Yaskawa INFORM job: DEMO_ROOF_UPPER_0625_3PAINT_45.JBI

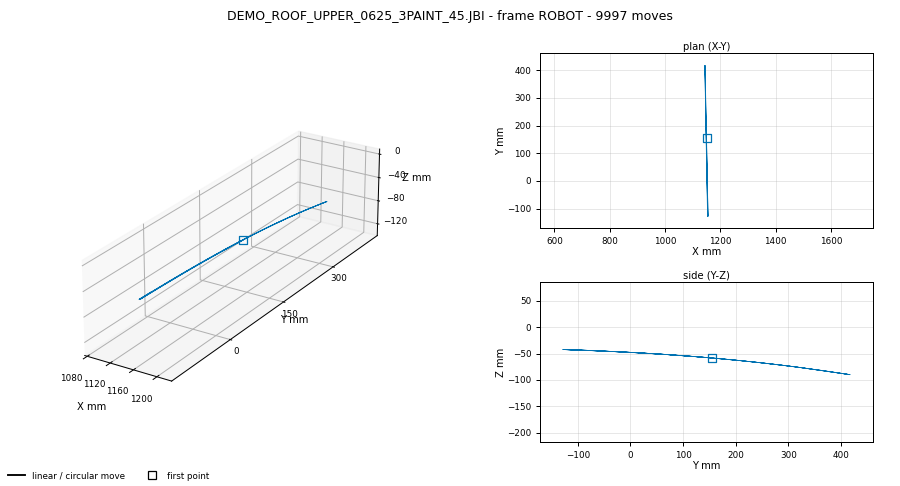
[picture p0: tool path of DEMO_ROOF_UPPER_0625_3PAINT_45.JBI in frame ROBOT, 9997 of 9997 moves have a stored position in this frame; points joined in program order, loops and branches not executed]
/JOB
//NAME DEMO_ROOF_UPPER_0625_3PAINT45
//POS
///NPOS 9997,0,0,0,0,0
///TOOL 0
///USER 0
///POSTYPE ROBOT
///RECTAN
///RCONF 1,0,0,0,0,0,0,0,0,0,0,0,0,0,0,0,0,0,0,0,0,0,0,0
C00000=1150.383,154.481,-58.197,-178.587,6.916,148.869
C00001=1150.389,154.232,-58.176,-178.590,6.914,148.870
C00002=1150.393,153.983,-58.154,-178.593,6.912,148.870
C00003=1150.398,153.733,-58.133,-178.596,6.910,148.870
C00004=1150.403,153.485,-58.111,-178.599,6.908,148.871
C00005=1150.407,153.236,-58.091,-178.601,6.907,148.871
C00006=1150.412,152.986,-58.069,-178.605,6.904,148.871
C00007=1150.417,152.737,-58.048,-178.607,6.902,148.872
C00008=1150.422,152.489,-58.026,-178.609,6.900,148.872
C00009=1150.426,152.240,-58.006,-178.612,6.899,148.872
C00010=1150.431,151.991,-57.984,-178.615,6.897,148.873
C00011=1150.436,151.741,-57.963,-178.618,6.894,148.873
C00012=1150.440,151.492,-57.941,-178.621,6.893,148.873
C00013=1150.445,151.243,-57.921,-178.624,6.891,148.874
C00014=1150.450,150.994,-57.900,-178.626,6.889,148.874
C00015=1150.455,150.745,-57.878,-178.629,6.887,148.875
C00016=1150.459,150.496,-57.857,-178.632,6.885,148.875
C00017=1150.464,150.247,-57.836,-178.635,6.883,148.875
C00018=1150.469,149.998,-57.815,-178.637,6.881,148.876
C00019=1150.473,149.749,-57.794,-178.640,6.879,148.876
C00020=1150.478,149.500,-57.773,-178.643,6.878,148.876
C00021=1150.483,149.251,-57.752,-178.645,6.876,148.877
C00022=1150.487,149.001,-57.731,-178.649,6.873,148.877
C00023=1150.492,148.752,-57.710,-178.651,6.872,148.877
C00024=1150.497,148.504,-57.688,-178.654,6.870,148.878
C00025=1150.502,148.255,-57.668,-178.657,6.868,148.878
C00026=1150.507,148.005,-57.647,-178.659,6.867,148.879
C00027=1150.511,147.756,-57.626,-178.662,6.865,148.879
C00028=1150.516,147.508,-57.605,-178.665,6.862,148.879
C00029=1150.521,147.258,-57.584,-178.668,6.860,148.879
C00030=1150.525,147.009,-57.563,-178.670,6.858,148.880
C00031=1150.530,146.760,-57.542,-178.673,6.857,148.880
C00032=1150.535,146.511,-57.522,-178.676,6.855,148.881
C00033=1150.540,146.262,-57.500,-178.679,6.853,148.881
C00034=1150.544,146.013,-57.480,-178.681,6.852,148.881
C00035=1150.549,145.764,-57.459,-178.685,6.849,148.882
C00036=1150.554,145.515,-57.438,-178.687,6.847,148.882
C00037=1150.559,145.266,-57.417,-178.690,6.846,148.883
C00038=1150.563,145.017,-57.397,-178.693,6.844,148.883
C00039=1150.568,144.767,-57.376,-178.695,6.842,148.883
C00040=1150.572,144.519,-57.355,-178.698,6.840,148.884
C00041=1150.577,144.269,-57.334,-178.701,6.839,148.884
C00042=1150.581,144.020,-57.313,-178.704,6.836,148.884
C00043=1150.587,143.771,-57.292,-178.707,6.835,148.885
C00044=1150.591,143.522,-57.272,-178.709,6.833,148.885
C00045=1150.596,143.273,-57.251,-178.712,6.831,148.885
C00046=1150.601,143.024,-57.231,-178.714,6.829,148.886
C00047=1150.606,142.774,-57.210,-178.717,6.827,148.886
C00048=1150.610,142.525,-57.189,-178.720,6.826,148.887
C00049=1150.616,142.276,-57.168,-178.723,6.823,148.887
C00050=1150.620,142.027,-57.148,-178.726,6.821,148.887
C00051=1150.624,141.778,-57.128,-178.729,6.820,148.888
C00052=1150.630,141.529,-57.107,-178.731,6.818,148.888
C00053=1150.634,141.280,-57.086,-178.734,6.816,148.889
C00054=1150.639,141.031,-57.065,-178.737,6.814,148.889
C00055=1150.644,140.782,-57.045,-178.739,6.813,148.889
C00056=1150.648,140.532,-57.025,-178.742,6.811,148.890
C00057=1150.654,140.283,-57.004,-178.745,6.809,148.890
C00058=1150.658,140.034,-56.984,-178.748,6.807,148.890
C00059=1150.662,139.785,-56.963,-178.751,6.805,148.891
C00060=1150.668,139.536,-56.943,-178.754,6.803,148.891
C00061=1150.672,139.287,-56.922,-178.756,6.802,148.892
C00062=1150.676,139.038,-56.902,-178.759,6.800,148.892
C00063=1150.682,138.789,-56.881,-178.762,6.798,148.892
C00064=1150.686,138.539,-56.861,-178.764,6.796,148.893
C00065=1150.691,138.290,-56.841,-178.767,6.795,148.893
C00066=1150.696,138.041,-56.820,-178.770,6.793,148.894
C00067=1150.700,137.792,-56.799,-178.773,6.791,148.894
C00068=1150.705,137.544,-56.779,-178.775,6.790,148.894
C00069=1150.710,137.294,-56.760,-178.779,6.787,148.895
C00070=1150.715,137.045,-56.739,-178.781,6.785,148.895
C00071=1150.720,136.796,-56.718,-178.784,6.784,148.895
C00072=1150.724,136.547,-56.698,-178.787,6.782,148.896
C00073=1150.729,136.297,-56.678,-178.789,6.780,148.896
C00074=1150.734,136.048,-56.657,-178.792,6.779,148.897
C00075=1150.739,135.799,-56.637,-178.795,6.777,148.897
C00076=1150.743,135.550,-56.617,-178.798,6.775,148.897
C00077=1150.748,135.301,-56.597,-178.800,6.773,148.898
C00078=1150.754,135.052,-56.576,-178.803,6.772,148.898
C00079=1150.758,134.803,-56.557,-178.806,6.770,148.899
C00080=1150.763,134.554,-56.536,-178.808,6.768,148.899
C00081=1150.767,134.305,-56.516,-178.811,6.767,148.899
C00082=1150.772,134.055,-56.496,-178.814,6.765,148.900
C00083=1150.776,133.806,-56.476,-178.817,6.762,148.900
C00084=1150.782,133.556,-56.456,-178.820,6.761,148.901
C00085=1150.787,133.308,-56.436,-178.823,6.759,148.901
C00086=1150.791,133.059,-56.415,-178.825,6.757,148.901
C00087=1150.796,132.810,-56.396,-178.828,6.755,148.902
C00088=1150.800,132.561,-56.375,-178.831,6.754,148.902
C00089=1150.805,132.311,-56.356,-178.833,6.752,148.903
C00090=1150.811,132.043,-56.333,-178.836,6.750,148.903
C00091=1150.815,131.774,-56.312,-178.839,6.749,148.904
C00092=1150.821,131.505,-56.291,-178.843,6.746,148.904
C00093=1150.826,131.237,-56.269,-178.845,6.745,148.904
C00094=1150.831,130.988,-56.249,-178.848,6.743,148.905
C00095=1150.836,130.739,-56.229,-178.851,6.741,148.905
C00096=1150.840,130.490,-56.209,-178.853,6.740,148.906
C00097=1150.845,130.240,-56.190,-178.856,6.738,148.906
C00098=1150.849,129.991,-56.169,-178.859,6.736,148.906
C00099=1150.856,129.742,-56.149,-178.862,6.734,148.907
C00100=1150.860,129.493,-56.129,-178.864,6.733,148.907
C00101=1150.865,129.243,-56.109,-178.867,6.731,148.907
C00102=1150.869,128.994,-56.090,-178.870,6.729,148.908
C00103=1150.874,128.746,-56.070,-178.872,6.728,148.908
C00104=1150.879,128.496,-56.050,-178.875,6.726,148.909
C00105=1150.884,128.247,-56.030,-178.878,6.724,148.909
C00106=1150.888,127.998,-56.010,-178.881,6.723,148.909
C00107=1150.894,127.749,-55.991,-178.884,6.721,148.910
C00108=1150.898,127.500,-55.970,-178.887,6.719,148.910
C00109=1150.903,127.250,-55.951,-178.889,6.718,148.911
C00110=1150.908,127.001,-55.931,-178.892,6.716,148.911
C00111=1150.912,126.752,-55.912,-178.895,6.714,148.912
C00112=1150.917,126.503,-55.892,-178.897,6.713,148.912
C00113=1150.921,126.254,-55.872,-178.900,6.711,148.912
C00114=1150.927,126.005,-55.853,-178.903,6.709,148.913
C00115=1150.931,125.756,-55.833,-178.906,6.708,148.913
C00116=1150.936,125.506,-55.813,-178.908,6.706,148.914
C00117=1150.941,125.257,-55.793,-178.911,6.704,148.914
C00118=1150.946,125.008,-55.774,-178.914,6.702,148.914
C00119=1150.951,124.758,-55.754,-178.916,6.701,148.915
C00120=1150.955,124.509,-55.734,-178.919,6.699,148.915
C00121=1150.961,124.260,-55.715,-178.922,6.698,148.916
C00122=1150.965,124.011,-55.696,-178.925,6.696,148.916
C00123=1150.969,123.762,-55.676,-178.928,6.694,148.917
C00124=1150.975,123.513,-55.657,-178.931,6.693,148.917
C00125=1150.979,123.263,-55.637,-178.933,6.691,148.917
C00126=1150.984,123.014,-55.617,-178.936,6.689,148.918
C00127=1150.989,122.765,-55.598,-178.939,6.687,148.918
C00128=1150.993,122.516,-55.578,-178.941,6.686,148.919
C00129=1150.999,122.267,-55.559,-178.944,6.684,148.919
C00130=1151.003,122.018,-55.540,-178.947,6.682,148.919
C00131=1151.008,121.768,-55.520,-178.950,6.681,148.920
C00132=1151.013,121.519,-55.501,-178.953,6.679,148.920
C00133=1151.017,121.270,-55.481,-178.955,6.678,148.921
C00134=1151.022,121.020,-55.462,-178.958,6.676,148.921
C00135=1151.027,120.771,-55.443,-178.961,6.674,148.922
C00136=1151.032,120.522,-55.423,-178.964,6.672,148.922
C00137=1151.037,120.273,-55.404,-178.966,6.671,148.923
C00138=1151.042,120.024,-55.385,-178.969,6.669,148.923
C00139=1151.047,119.775,-55.365,-178.972,6.667,148.923
C00140=1151.052,119.525,-55.346,-178.974,6.666,148.924
C00141=1151.056,119.276,-55.327,-178.977,6.664,148.924
C00142=1151.061,119.027,-55.307,-178.980,6.663,148.925
C00143=1151.066,118.778,-55.288,-178.983,6.662,148.925
C00144=1151.071,118.529,-55.268,-178.985,6.660,148.926
C00145=1151.075,118.280,-55.249,-178.988,6.658,148.926
C00146=1151.080,118.031,-55.230,-178.991,6.657,148.926
C00147=1151.085,117.781,-55.210,-178.993,6.655,148.927
C00148=1151.090,117.533,-55.192,-178.996,6.653,148.927
C00149=1151.095,117.282,-55.173,-178.999,6.651,148.928
C00150=1151.100,117.033,-55.153,-179.002,6.650,148.928
C00151=1151.104,116.784,-55.134,-179.005,6.648,148.929
C00152=1151.109,116.535,-55.115,-179.008,6.647,148.929
C00153=1151.114,116.286,-55.095,-179.010,6.645,148.929
C00154=1151.118,116.037,-55.076,-179.013,6.643,148.930
C00155=1151.124,115.787,-55.058,-179.016,6.642,148.930
C00156=1151.129,115.537,-55.038,-179.018,6.640,148.931
C00157=1151.133,115.289,-55.019,-179.021,6.639,148.931
C00158=1151.138,115.039,-55.000,-179.024,6.638,148.932
C00159=1151.143,114.791,-54.981,-179.026,6.636,148.932
C00160=1151.148,114.541,-54.962,-179.029,6.634,148.932
C00161=1151.153,114.292,-54.943,-179.032,6.633,148.933
C00162=1151.158,114.043,-54.924,-179.035,6.631,148.933
C00163=1151.162,113.794,-54.904,-179.037,6.629,148.934
C00164=1151.167,113.544,-54.886,-179.040,6.627,148.934
C00165=1151.172,113.295,-54.867,-179.043,6.626,148.935
C00166=1151.177,113.046,-54.848,-179.046,6.624,148.935
C00167=1151.182,112.796,-54.829,-179.049,6.623,148.936
C00168=1151.186,112.548,-54.810,-179.051,6.622,148.936
C00169=1151.191,112.298,-54.791,-179.054,6.620,148.936
C00170=1151.196,112.049,-54.773,-179.056,6.618,148.937
C00171=1151.201,111.800,-54.754,-179.059,6.617,148.937
C00172=1151.206,111.550,-54.734,-179.062,6.615,148.938
C00173=1151.211,111.301,-54.716,-179.065,6.614,148.938
C00174=1151.215,111.052,-54.697,-179.068,6.612,148.939
C00175=1151.221,110.802,-54.678,-179.070,6.610,148.939
C00176=1151.225,110.554,-54.660,-179.073,6.609,148.939
C00177=1151.230,110.304,-54.640,-179.075,6.608,148.940
C00178=1151.235,110.055,-54.622,-179.078,6.606,148.940
C00179=1151.240,109.806,-54.602,-179.081,6.605,148.941
C00180=1151.245,109.556,-54.584,-179.084,6.603,148.941
C00181=1151.250,109.308,-54.565,-179.087,6.601,148.942
C00182=1151.254,109.058,-54.547,-179.089,6.600,148.942
C00183=1151.260,108.809,-54.527,-179.092,6.598,148.943
C00184=1151.264,108.559,-54.509,-179.095,6.597,148.943
C00185=1151.268,108.310,-54.490,-179.097,6.596,148.944
C00186=1151.274,108.061,-54.472,-179.100,6.594,148.944
C00187=1151.278,107.812,-54.453,-179.103,6.592,148.944
C00188=1151.283,107.562,-54.435,-179.106,6.591,148.945
C00189=1151.288,107.314,-54.415,-179.108,6.589,148.945
C00190=1151.293,107.064,-54.397,-179.112,6.588,148.946
C00191=1151.298,106.814,-54.379,-179.114,6.586,148.946
C00192=1151.303,106.566,-54.360,-179.116,6.585,148.947
C00193=1151.307,106.316,-54.341,-179.119,6.583,148.947
C00194=1151.313,106.048,-54.321,-179.122,6.582,148.947
C00195=1151.318,105.780,-54.301,-179.125,6.580,148.948
C00196=1151.324,105.511,-54.281,-179.128,6.579,148.949
C00197=1151.328,105.242,-54.262,-179.132,6.576,148.949
C00198=1151.333,104.993,-54.242,-179.134,6.576,148.950
C00199=1151.338,104.744,-54.224,-179.136,6.574,148.950
C00200=1151.343,104.495,-54.206,-179.139,6.572,148.950
C00201=1151.347,104.246,-54.187,-179.142,6.571,148.951
C00202=1151.353,103.996,-54.169,-179.145,6.569,148.951
C00203=1151.358,103.747,-54.151,-179.148,6.568,148.952
C00204=1151.362,103.498,-54.132,-179.150,6.567,148.952
C00205=1151.367,103.248,-54.114,-179.153,6.565,148.953
C00206=1151.372,102.999,-54.095,-179.155,6.563,148.953
C00207=1151.377,102.750,-54.077,-179.159,6.562,148.954
C00208=1151.381,102.501,-54.058,-179.161,6.560,148.954
C00209=1151.386,102.251,-54.040,-179.164,6.559,148.955
C00210=1151.392,102.002,-54.021,-179.166,6.558,148.955
C00211=1151.397,101.753,-54.003,-179.169,6.556,148.955
C00212=1151.402,101.504,-53.986,-179.172,6.555,148.956
C00213=1151.406,101.254,-53.966,-179.175,6.553,148.956
C00214=1151.411,101.005,-53.948,-179.178,6.551,148.957
C00215=1151.416,100.756,-53.930,-179.180,6.550,148.957
C00216=1151.421,100.506,-53.912,-179.182,6.549,148.958
C00217=1151.426,100.257,-53.894,-179.186,6.547,148.958
C00218=1151.430,100.007,-53.876,-179.188,6.546,148.959
C00219=1151.435,99.758,-53.858,-179.191,6.544,148.959
C00220=1151.440,99.510,-53.839,-179.193,6.543,148.960
C00221=1151.446,99.260,-53.820,-179.196,6.541,148.960
C00222=1151.450,99.010,-53.802,-179.199,6.540,148.961
C00223=1151.455,98.761,-53.784,-179.202,6.538,148.961
C00224=1151.460,98.512,-53.766,-179.205,6.537,148.961
C00225=1151.465,98.263,-53.748,-179.207,6.536,148.962
C00226=1151.470,98.014,-53.730,-179.210,6.534,148.963
C00227=1151.474,97.764,-53.712,-179.213,6.533,148.963
C00228=1151.479,97.515,-53.694,-179.216,6.531,148.963
C00229=1151.484,97.265,-53.676,-179.218,6.529,148.964
C00230=1151.489,97.016,-53.658,-179.221,6.529,148.964
C00231=1151.494,96.767,-53.639,-179.224,6.527,148.965
C00232=1151.499,96.518,-53.621,-179.226,6.526,148.965
C00233=1151.504,96.268,-53.603,-179.229,6.524,148.966
C00234=1151.509,96.019,-53.585,-179.231,6.523,148.966
C00235=1151.513,95.769,-53.567,-179.234,6.522,148.967
C00236=1151.518,95.520,-53.549,-179.237,6.520,148.967
C00237=1151.523,95.271,-53.531,-179.240,6.518,148.968
C00238=1151.528,95.022,-53.513,-179.243,6.517,148.968
C00239=1151.533,94.773,-53.495,-179.245,6.516,148.969
C00240=1151.538,94.523,-53.477,-179.248,6.514,148.969
C00241=1151.543,94.274,-53.459,-179.251,6.513,148.969
C00242=1151.548,94.024,-53.442,-179.253,6.511,148.970
C00243=1151.553,93.775,-53.424,-179.256,6.511,148.971
C00244=1151.558,93.526,-53.406,-179.259,6.509,148.971
C00245=1151.563,93.277,-53.388,-179.261,6.507,148.971
C00246=1151.567,93.027,-53.370,-179.264,6.505,148.972
C00247=1151.572,92.778,-53.352,-179.267,6.505,148.972
C00248=1151.577,92.528,-53.334,-179.270,6.503,148.973
C00249=1151.582,92.279,-53.316,-179.272,6.502,148.973
C00250=1151.587,92.030,-53.298,-179.275,6.500,148.974
C00251=1151.591,91.781,-53.281,-179.278,6.499,148.974
C00252=1151.596,91.532,-53.263,-179.280,6.498,148.975
C00253=1151.601,91.282,-53.246,-179.283,6.496,148.975
C00254=1151.606,91.033,-53.228,-179.286,6.494,148.976
C00255=1151.611,90.784,-53.210,-179.288,6.494,148.976
C00256=1151.616,90.534,-53.192,-179.291,6.492,148.977
C00257=1151.621,90.285,-53.174,-179.294,6.490,148.977
C00258=1151.626,90.035,-53.156,-179.297,6.489,148.978
C00259=1151.631,89.786,-53.139,-179.299,6.488,148.978
C00260=1151.636,89.537,-53.122,-179.302,6.487,148.979
C00261=1151.640,89.288,-53.104,-179.305,6.485,148.979
C00262=1151.645,89.038,-53.086,-179.307,6.484,148.980
C00263=1151.650,88.789,-53.068,-179.310,6.483,148.980
C00264=1151.656,88.539,-53.051,-179.313,6.481,148.980
C00265=1151.660,88.290,-53.033,-179.316,6.479,148.981
C00266=1151.665,88.041,-53.016,-179.318,6.479,148.982
C00267=1151.670,87.792,-52.998,-179.321,6.477,148.982
C00268=1151.675,87.542,-52.980,-179.324,6.475,148.982
C00269=1151.680,87.293,-52.963,-179.327,6.474,148.983
C00270=1151.685,87.043,-52.945,-179.329,6.473,148.983
C00271=1151.689,86.794,-52.928,-179.332,6.472,148.984
C00272=1151.694,86.545,-52.910,-179.335,6.470,148.984
C00273=1151.699,86.296,-52.892,-179.337,6.469,148.985
C00274=1151.704,86.046,-52.875,-179.340,6.468,148.985
C00275=1151.709,85.797,-52.858,-179.343,6.466,148.986
C00276=1151.714,85.547,-52.840,-179.345,6.465,148.986
C00277=1151.719,85.298,-52.822,-179.348,6.464,148.987
C00278=1151.725,85.049,-52.805,-179.351,6.462,148.987
C00279=1151.729,84.800,-52.788,-179.353,6.460,148.988
C00280=1151.734,84.550,-52.771,-179.356,6.460,148.988
C00281=1151.739,84.301,-52.753,-179.359,6.458,148.989
C00282=1151.744,84.051,-52.735,-179.362,6.457,148.989
C00283=1151.748,83.802,-52.718,-179.364,6.456,148.990
C00284=1151.753,83.553,-52.701,-179.367,6.454,148.990
C00285=1151.758,83.303,-52.683,-179.370,6.453,148.991
C00286=1151.763,83.054,-52.666,-179.372,6.452,148.991
C00287=1151.768,82.804,-52.649,-179.375,6.451,148.992
C00288=1151.774,82.556,-52.631,-179.378,6.449,148.992
C00289=1151.778,82.306,-52.615,-179.380,6.448,148.993
C00290=1151.783,82.057,-52.597,-179.383,6.447,148.993
C00291=1151.788,81.807,-52.579,-179.386,6.445,148.994
C00292=1151.793,81.558,-52.563,-179.388,6.444,148.994
C00293=1151.798,81.309,-52.545,-179.391,6.443,148.995
C00294=1151.802,81.059,-52.528,-179.394,6.441,148.995
C00295=1151.808,80.810,-52.511,-179.396,6.440,148.996
C00296=1151.813,80.561,-52.493,-179.399,6.439,148.996
C00297=1151.817,80.311,-52.477,-179.402,6.437,148.997
C00298=1151.823,80.042,-52.458,-179.405,6.436,148.997
C00299=1151.829,79.774,-52.439,-179.408,6.434,148.998
C00300=1151.833,79.506,-52.421,-179.410,6.433,148.998
C00301=1151.838,79.237,-52.402,-179.413,6.432,148.999
C00302=1151.843,78.989,-52.386,-179.416,6.431,148.999
C00303=1151.849,78.739,-52.368,-179.419,6.429,149.000
C00304=1151.854,78.489,-52.351,-179.421,6.428,149.000
C00305=1151.858,78.240,-52.334,-179.424,6.427,149.001
C00306=1151.863,77.990,-52.317,-179.426,6.426,149.001
C00307=1151.868,77.742,-52.300,-179.430,6.424,149.002
C00308=1151.874,77.492,-52.283,-179.432,6.423,149.002
C00309=1151.878,77.243,-52.266,-179.434,6.422,149.003
C00310=1151.883,76.993,-52.248,-179.438,6.421,149.003
C00311=1151.887,76.744,-52.232,-179.440,6.419,149.004
C00312=1151.893,76.495,-52.215,-179.443,6.418,149.004
C00313=1151.898,76.245,-52.198,-179.446,6.417,149.005
C00314=1151.903,75.995,-52.181,-179.449,6.415,149.005
C00315=1151.907,75.746,-52.164,-179.451,6.414,149.006
C00316=1151.913,75.497,-52.147,-179.453,6.413,149.006
C00317=1151.917,75.248,-52.130,-179.456,6.412,149.007
C00318=1151.923,74.998,-52.113,-179.459,6.410,149.007
C00319=1151.927,74.749,-52.096,-179.462,6.409,149.008
C00320=1151.932,74.500,-52.080,-179.464,6.408,149.008
C00321=1151.937,74.250,-52.062,-179.467,6.407,149.009
C00322=1151.942,74.001,-52.046,-179.470,6.405,149.009
C00323=1151.948,73.751,-52.029,-179.472,6.404,149.010
C00324=1151.952,73.502,-52.012,-179.475,6.403,149.010
C00325=1151.957,73.252,-51.995,-179.477,6.402,149.011
C00326=1151.962,73.003,-51.978,-179.480,6.401,149.011
C00327=1151.967,72.754,-51.962,-179.483,6.399,149.012
C00328=1151.972,72.504,-51.945,-179.486,6.398,149.013
C00329=1151.977,72.255,-51.928,-179.489,6.397,149.013
C00330=1151.982,72.006,-51.912,-179.491,6.396,149.013
C00331=1151.987,71.756,-51.894,-179.494,6.395,149.014
C00332=1151.991,71.507,-51.878,-179.497,6.393,149.014
C00333=1151.997,71.258,-51.861,-179.499,6.392,149.015
C00334=1152.002,71.008,-51.844,-179.502,6.391,149.016
C00335=1152.006,70.759,-51.827,-179.504,6.390,149.016
C00336=1152.011,70.510,-51.811,-179.507,6.388,149.016
C00337=1152.017,70.260,-51.794,-179.510,6.387,149.017
C00338=1152.021,70.010,-51.777,-179.512,6.386,149.017
C00339=1152.026,69.762,-51.761,-179.515,6.384,149.018
C00340=1152.031,69.512,-51.744,-179.518,6.384,149.019
C00341=1152.036,69.262,-51.728,-179.520,6.382,149.019
C00342=1152.041,69.013,-51.711,-179.523,6.381,149.019
C00343=1152.046,68.763,-51.694,-179.526,6.380,149.020
C00344=1152.051,68.514,-51.678,-179.529,6.378,149.021
C00345=1152.056,68.265,-51.661,-179.531,6.378,149.021
C00346=1152.060,68.015,-51.644,-179.534,6.376,149.022
C00347=1152.067,67.766,-51.628,-179.536,6.375,149.022
C00348=1152.071,67.516,-51.612,-179.539,6.374,149.023
C00349=1152.076,67.267,-51.595,-179.542,6.372,149.023
C00350=1152.081,67.018,-51.579,-179.544,6.372,149.024
C00351=1152.086,66.768,-51.561,-179.547,6.370,149.024
C00352=1152.091,66.519,-51.546,-179.550,6.369,149.025
C00353=1152.096,66.269,-51.529,-179.552,6.368,149.025
C00354=1152.100,66.020,-51.512,-179.555,6.367,149.026
C00355=1152.105,65.771,-51.496,-179.558,6.366,149.026
C00356=1152.111,65.521,-51.480,-179.560,6.364,149.027
C00357=1152.116,65.272,-51.463,-179.563,6.363,149.027
C00358=1152.120,65.022,-51.447,-179.566,6.362,149.028
C00359=1152.125,64.774,-51.430,-179.568,6.361,149.028
C00360=1152.130,64.523,-51.414,-179.571,6.360,149.029
C00361=1152.135,64.275,-51.398,-179.573,6.359,149.029
C00362=1152.140,64.025,-51.381,-179.577,6.357,149.030
C00363=1152.145,63.775,-51.365,-179.579,6.357,149.030
C00364=1152.150,63.526,-51.349,-179.581,6.355,149.031
C00365=1152.155,63.276,-51.333,-179.585,6.354,149.031
C00366=1152.160,63.027,-51.316,-179.587,6.353,149.032
C00367=1152.165,62.778,-51.300,-179.590,6.351,149.032
C00368=1152.170,62.528,-51.284,-179.592,6.351,149.033
C00369=1152.175,62.279,-51.267,-179.595,6.349,149.033
C00370=1152.180,62.030,-51.251,-179.598,6.348,149.034
C00371=1152.185,61.780,-51.235,-179.600,6.347,149.035
C00372=1152.190,61.531,-51.218,-179.602,6.346,149.035
C00373=1152.195,61.281,-51.202,-179.606,6.345,149.036
C00374=1152.200,61.032,-51.186,-179.608,6.344,149.036
C00375=1152.205,60.782,-51.170,-179.611,6.342,149.037
C00376=1152.210,60.533,-51.154,-179.613,6.342,149.037
C00377=1152.215,60.283,-51.138,-179.616,6.340,149.038
C00378=1152.220,60.034,-51.121,-179.619,6.339,149.038
C00379=1152.225,59.784,-51.105,-179.621,6.338,149.039
C00380=1152.230,59.535,-51.089,-179.624,6.336,149.039
C00381=1152.235,59.286,-51.074,-179.627,6.336,149.040
C00382=1152.240,59.036,-51.057,-179.629,6.334,149.040
C00383=1152.245,58.787,-51.041,-179.632,6.334,149.041
C00384=1152.249,58.537,-51.025,-179.635,6.332,149.041
C00385=1152.255,58.288,-51.009,-179.637,6.331,149.042
C00386=1152.259,58.039,-50.992,-179.640,6.330,149.042
C00387=1152.265,57.789,-50.977,-179.642,6.329,149.043
C00388=1152.270,57.539,-50.961,-179.646,6.328,149.044
C00389=1152.275,57.290,-50.945,-179.648,6.327,149.044
C00390=1152.280,57.041,-50.929,-179.651,6.325,149.044
C00391=1152.284,56.791,-50.912,-179.653,6.325,149.045
C00392=1152.290,56.542,-50.897,-179.656,6.323,149.046
C00393=1152.295,56.292,-50.881,-179.658,6.322,149.046
C00394=1152.300,56.043,-50.864,-179.661,6.321,149.047
C00395=1152.305,55.794,-50.849,-179.663,6.320,149.047
C00396=1152.310,55.544,-50.833,-179.667,6.319,149.048
C00397=1152.315,55.295,-50.817,-179.669,6.318,149.048
C00398=1152.319,55.045,-50.801,-179.672,6.316,149.049
C00399=1152.324,54.796,-50.786,-179.674,6.316,149.049
C00400=1152.329,54.547,-50.769,-179.677,6.314,149.050
C00401=1152.334,54.297,-50.753,-179.680,6.313,149.050
C00402=1152.340,54.028,-50.736,-179.682,6.312,149.051
C00403=1152.345,53.760,-50.719,-179.685,6.311,149.052
C00404=1152.351,53.491,-50.702,-179.688,6.310,149.052
C00405=1152.356,53.223,-50.685,-179.691,6.308,149.053
C00406=1152.361,52.973,-50.669,-179.693,6.308,149.053
C00407=1152.367,52.723,-50.654,-179.696,6.306,149.054
C00408=1152.371,52.475,-50.638,-179.699,6.305,149.054
C00409=1152.376,52.225,-50.622,-179.702,6.304,149.055
C00410=1152.381,51.975,-50.607,-179.704,6.303,149.055
C00411=1152.387,51.726,-50.591,-179.706,6.302,149.056
C00412=1152.391,51.476,-50.575,-179.709,6.301,149.056
C00413=1152.396,51.227,-50.559,-179.711,6.300,149.057
C00414=1152.401,50.978,-50.544,-179.715,6.299,149.058
C00415=1152.406,50.728,-50.528,-179.717,6.298,149.058
C00416=1152.411,50.478,-50.512,-179.720,6.297,149.058
C00417=1152.417,50.229,-50.497,-179.722,6.296,149.059
C00418=1152.421,49.979,-50.481,-179.725,6.294,149.060
C00419=1152.426,49.730,-50.466,-179.728,6.294,149.060
C00420=1152.431,49.481,-50.449,-179.730,6.292,149.061
C00421=1152.437,49.232,-50.434,-179.733,6.292,149.061
C00422=1152.441,48.982,-50.418,-179.735,6.291,149.062
C00423=1152.446,48.732,-50.403,-179.738,6.289,149.062
C00424=1152.451,48.483,-50.387,-179.741,6.289,149.063
C00425=1152.456,48.233,-50.371,-179.743,6.287,149.063
C00426=1152.461,47.984,-50.356,-179.746,6.287,149.064
C00427=1152.466,47.734,-50.341,-179.749,6.285,149.064
C00428=1152.472,47.485,-50.325,-179.751,6.284,149.065
C00429=1152.476,47.235,-50.310,-179.754,6.283,149.066
C00430=1152.481,46.986,-50.294,-179.756,6.282,149.066
C00431=1152.486,46.736,-50.279,-179.759,6.282,149.067
C00432=1152.491,46.487,-50.264,-179.762,6.280,149.067
C00433=1152.496,46.238,-50.248,-179.764,6.279,149.068
C00434=1152.501,45.988,-50.232,-179.767,6.278,149.068
C00435=1152.506,45.739,-50.217,-179.769,6.277,149.069
C00436=1152.511,45.489,-50.201,-179.772,6.276,149.069
C00437=1152.517,45.240,-50.186,-179.775,6.275,149.070
C00438=1152.521,44.990,-50.171,-179.777,6.274,149.070
C00439=1152.526,44.741,-50.155,-179.780,6.273,149.071
C00440=1152.531,44.491,-50.139,-179.783,6.272,149.072
C00441=1152.536,44.242,-50.124,-179.785,6.271,149.072
C00442=1152.541,43.993,-50.109,-179.788,6.270,149.072
C00443=1152.546,43.742,-50.094,-179.790,6.269,149.073
C00444=1152.551,43.493,-50.079,-179.793,6.268,149.074
C00445=1152.557,43.244,-50.063,-179.796,6.267,149.074
C00446=1152.561,42.995,-50.048,-179.798,6.265,149.075
C00447=1152.567,42.745,-50.032,-179.801,6.265,149.075
C00448=1152.571,42.496,-50.017,-179.803,6.264,149.076
C00449=1152.576,42.246,-50.001,-179.806,6.262,149.076
C00450=1152.582,41.996,-49.987,-179.809,6.262,149.077
C00451=1152.586,41.747,-49.972,-179.811,6.260,149.077
C00452=1152.592,41.497,-49.956,-179.814,6.260,149.078
C00453=1152.596,41.248,-49.941,-179.816,6.259,149.078
C00454=1152.602,40.999,-49.925,-179.819,6.258,149.079
C00455=1152.607,40.749,-49.911,-179.821,6.257,149.080
C00456=1152.612,40.499,-49.895,-179.825,6.256,149.080
C00457=1152.616,40.250,-49.880,-179.827,6.255,149.081
C00458=1152.622,40.001,-49.865,-179.829,6.254,149.081
C00459=1152.627,39.751,-49.850,-179.832,6.253,149.082
C00460=1152.632,39.502,-49.835,-179.834,6.252,149.082
C00461=1152.637,39.252,-49.820,-179.838,6.251,149.083
C00462=1152.642,39.003,-49.804,-179.840,6.250,149.083
C00463=1152.647,38.753,-49.790,-179.842,6.249,149.084
C00464=1152.652,38.504,-49.774,-179.845,6.248,149.085
C00465=1152.657,38.255,-49.759,-179.847,6.247,149.085
C00466=1152.662,38.004,-49.744,-179.850,6.246,149.086
C00467=1152.667,37.755,-49.729,-179.853,6.245,149.086
C00468=1152.672,37.506,-49.713,-179.855,6.244,149.087
C00469=1152.677,37.256,-49.699,-179.858,6.243,149.087
C00470=1152.682,37.006,-49.684,-179.861,6.242,149.088
C00471=1152.687,36.757,-49.669,-179.863,6.241,149.088
C00472=1152.692,36.508,-49.654,-179.866,6.240,149.089
C00473=1152.697,36.258,-49.639,-179.868,6.239,149.089
C00474=1152.702,36.009,-49.624,-179.871,6.238,149.090
C00475=1152.708,35.759,-49.609,-179.874,6.237,149.091
C00476=1152.713,35.509,-49.595,-179.876,6.236,149.091
C00477=1152.717,35.260,-49.580,-179.879,6.236,149.092
C00478=1152.723,35.011,-49.564,-179.881,6.234,149.092
C00479=1152.728,34.761,-49.550,-179.884,6.234,149.093
C00480=1152.733,34.512,-49.534,-179.886,6.233,149.093
C00481=1152.738,34.262,-49.520,-179.889,6.231,149.094
C00482=1152.743,34.013,-49.505,-179.892,6.231,149.094
C00483=1152.748,33.763,-49.490,-179.895,6.229,149.095
C00484=1152.753,33.514,-49.475,-179.897,6.229,149.096
C00485=1152.758,33.264,-49.461,-179.899,6.228,149.096
C00486=1152.763,33.015,-49.445,-179.902,6.226,149.097
C00487=1152.768,32.765,-49.431,-179.905,6.226,149.097
C00488=1152.773,32.516,-49.416,-179.907,6.225,149.098
C00489=1152.779,32.266,-49.401,-179.910,6.223,149.098
C00490=1152.783,32.017,-49.386,-179.913,6.223,149.099
C00491=1152.788,31.767,-49.372,-179.915,6.222,149.099
C00492=1152.793,31.518,-49.357,-179.918,6.221,149.100
C00493=1152.799,31.268,-49.342,-179.920,6.220,149.100
C00494=1152.804,31.018,-49.328,-179.923,6.220,149.101
C00495=1152.808,30.769,-49.313,-179.926,6.218,149.102
C00496=1152.814,30.519,-49.298,-179.928,6.217,149.102
C00497=1152.819,30.270,-49.283,-179.930,6.217,149.103
C00498=1152.824,30.020,-49.268,-179.933,6.216,149.103
C00499=1152.829,29.771,-49.254,-179.936,6.215,149.104
C00500=1152.834,29.521,-49.239,-179.938,6.214,149.104
C00501=1152.839,29.272,-49.224,-179.941,6.213,149.105
C00502=1152.844,29.022,-49.210,-179.943,6.212,149.105
C00503=1152.848,28.773,-49.195,-179.946,6.211,149.106
C00504=1152.854,28.524,-49.181,-179.948,6.210,149.107
C00505=1152.860,28.274,-49.166,-179.951,6.209,149.107
C00506=1152.865,28.005,-49.151,-179.954,6.208,149.108
C00507=1152.870,27.736,-49.135,-179.957,6.207,149.108
C00508=1152.876,27.467,-49.119,-179.959,6.207,149.109
C00509=1152.881,27.198,-49.103,-179.962,6.205,149.110
C00510=1152.886,26.949,-49.089,-179.965,6.204,149.110
C00511=1152.891,26.699,-49.074,-179.967,6.204,149.111
C00512=1152.896,26.449,-49.060,-179.970,6.202,149.111
C00513=1152.901,26.200,-49.044,-179.972,6.201,149.112
C00514=1152.907,25.951,-49.030,-179.975,6.201,149.112
C00515=1152.912,25.701,-49.016,-179.977,6.200,149.113
C00516=1152.917,25.451,-49.002,-179.980,6.199,149.113
C00517=1152.922,25.202,-48.988,-179.983,6.198,149.114
C00518=1152.926,24.953,-48.973,-179.985,6.197,149.115
C00519=1152.931,24.703,-48.958,-179.988,6.196,149.115
C00520=1152.936,24.453,-48.944,-179.990,6.195,149.116
C00521=1152.942,24.204,-48.930,-179.993,6.195,149.116
C00522=1152.947,23.954,-48.915,-179.995,6.194,149.117
C00523=1152.952,23.705,-48.900,-179.998,6.193,149.117
C00524=1152.957,23.455,-48.886,180.000,6.192,149.118
C00525=1152.962,23.206,-48.872,179.997,6.191,149.119
C00526=1152.967,22.956,-48.858,179.994,6.190,149.119
C00527=1152.972,22.706,-48.843,179.991,6.189,149.120
C00528=1152.977,22.457,-48.829,179.989,6.188,149.120
C00529=1152.982,22.207,-48.815,179.987,6.188,149.121
C00530=1152.987,21.958,-48.801,179.984,6.186,149.121
C00531=1152.992,21.708,-48.786,179.982,6.185,149.122
C00532=1152.997,21.458,-48.772,179.979,6.185,149.122
C00533=1153.003,21.210,-48.758,179.977,6.184,149.123
C00534=1153.007,20.960,-48.743,179.974,6.183,149.124
C00535=1153.012,20.711,-48.729,179.972,6.182,149.124
C00536=1153.017,20.461,-48.715,179.969,6.182,149.125
C00537=1153.022,20.211,-48.700,179.967,6.181,149.125
C00538=1153.028,19.962,-48.687,179.963,6.180,149.126
C00539=1153.033,19.712,-48.672,179.961,6.179,149.126
C00540=1153.038,19.463,-48.658,179.959,6.178,149.127
C00541=1153.043,19.213,-48.644,179.956,6.177,149.127
C00542=1153.048,18.964,-48.630,179.953,6.176,149.128
C00543=1153.053,18.714,-48.616,179.951,6.175,149.129
C00544=1153.058,18.465,-48.601,179.948,6.175,149.129
C00545=1153.063,18.215,-48.587,179.946,6.174,149.130
C00546=1153.069,17.966,-48.573,179.943,6.173,149.130
C00547=1153.074,17.715,-48.560,179.941,6.172,149.131
C00548=1153.079,17.466,-48.545,179.938,6.172,149.132
C00549=1153.084,17.216,-48.531,179.936,6.171,149.132
C00550=1153.089,16.967,-48.517,179.933,6.169,149.133
C00551=1153.094,16.717,-48.503,179.931,6.169,149.133
C00552=1153.099,16.468,-48.488,179.928,6.168,149.134
C00553=1153.104,16.218,-48.474,179.926,6.167,149.134
C00554=1153.110,15.969,-48.460,179.923,6.166,149.135
C00555=1153.114,15.720,-48.447,179.920,6.165,149.135
C00556=1153.119,15.470,-48.432,179.918,6.164,149.136
C00557=1153.125,15.220,-48.419,179.916,6.164,149.137
C00558=1153.130,14.970,-48.405,179.913,6.163,149.137
C00559=1153.135,14.721,-48.391,179.910,6.162,149.138
C00560=1153.140,14.472,-48.377,179.908,6.161,149.138
C00561=1153.145,14.222,-48.362,179.905,6.161,149.139
C00562=1153.150,13.973,-48.349,179.903,6.160,149.139
C00563=1153.155,13.723,-48.336,179.900,6.159,149.140
C00564=1153.160,13.473,-48.321,179.898,6.158,149.140
C00565=1153.165,13.224,-48.307,179.895,6.157,149.141
C00566=1153.171,12.975,-48.293,179.893,6.156,149.142
C00567=1153.176,12.724,-48.280,179.890,6.156,149.142
C00568=1153.180,12.475,-48.266,179.887,6.154,149.143
C00569=1153.186,12.226,-48.252,179.885,6.154,149.143
C00570=1153.191,11.976,-48.238,179.883,6.153,149.144
C00571=1153.196,11.726,-48.224,179.880,6.153,149.145
C00572=1153.202,11.477,-48.210,179.878,6.152,149.145
C00573=1153.206,11.227,-48.196,179.875,6.151,149.146
C00574=1153.211,10.977,-48.183,179.872,6.150,149.146
C00575=1153.217,10.728,-48.169,179.870,6.149,149.147
C00576=1153.222,10.478,-48.155,179.868,6.148,149.147
C00577=1153.227,10.229,-48.141,179.865,6.148,149.148
C00578=1153.232,9.979,-48.128,179.862,6.146,149.148
C00579=1153.237,9.730,-48.114,179.860,6.146,149.149
C00580=1153.242,9.481,-48.100,179.857,6.145,149.150
C00581=1153.247,9.231,-48.087,179.855,6.144,149.150
C00582=1153.252,8.982,-48.073,179.853,6.144,149.151
C00583=1153.258,8.731,-48.059,179.850,6.142,149.151
C00584=1153.263,8.482,-48.045,179.847,6.142,149.152
C00585=1153.267,8.233,-48.032,179.845,6.141,149.152
C00586=1153.273,7.982,-48.018,179.842,6.140,149.153
C00587=1153.278,7.733,-48.004,179.840,6.140,149.154
C00588=1153.283,7.483,-47.991,179.837,6.139,149.154
C00589=1153.288,7.234,-47.977,179.835,6.138,149.155
C00590=1153.293,6.985,-47.963,179.832,6.137,149.155
C00591=1153.298,6.735,-47.950,179.830,6.136,149.156
C00592=1153.303,6.486,-47.936,179.827,6.136,149.157
C00593=1153.309,6.235,-47.923,179.825,6.135,149.157
C00594=1153.313,5.987,-47.909,179.822,6.135,149.158
C00595=1153.319,5.736,-47.896,179.820,6.133,149.158
C00596=1153.324,5.487,-47.882,179.817,6.133,149.159
C00597=1153.329,5.237,-47.869,179.815,6.132,149.159
C00598=1153.334,4.988,-47.855,179.812,6.131,149.160
C00599=1153.340,4.738,-47.841,179.810,6.130,149.160
C00600=1153.344,4.489,-47.828,179.807,6.130,149.161
C00601=1153.350,4.239,-47.814,179.805,6.128,149.162
C00602=1153.354,3.990,-47.801,179.802,6.128,149.162
C00603=1153.360,3.740,-47.788,179.800,6.127,149.163
C00604=1153.365,3.490,-47.773,179.797,6.127,149.163
C00605=1153.370,3.241,-47.761,179.795,6.126,149.164
C00606=1153.375,2.991,-47.747,179.792,6.125,149.165
C00607=1153.380,2.742,-47.734,179.790,6.125,149.165
C00608=1153.385,2.492,-47.720,179.787,6.123,149.166
C00609=1153.391,2.243,-47.706,179.785,6.123,149.166
C00610=1153.396,1.973,-47.693,179.782,6.122,149.167
C00611=1153.401,1.703,-47.678,179.779,6.122,149.168
C00612=1153.407,1.434,-47.664,179.777,6.120,149.168
C00613=1153.412,1.165,-47.649,179.774,6.120,149.169
C00614=1153.418,0.915,-47.636,179.772,6.119,149.169
C00615=1153.422,0.666,-47.622,179.769,6.118,149.170
C00616=1153.428,0.416,-47.609,179.767,6.118,149.170
C00617=1153.433,0.166,-47.596,179.764,6.116,149.171
C00618=1153.438,-0.083,-47.582,179.761,6.115,149.171
C00619=1153.443,-0.333,-47.569,179.759,6.115,149.172
C00620=1153.449,-0.582,-47.556,179.757,6.114,149.173
C00621=1153.454,-0.832,-47.542,179.754,6.114,149.173
C00622=1153.459,-1.081,-47.529,179.752,6.113,149.174
C00623=1153.464,-1.331,-47.516,179.749,6.113,149.174
C00624=1153.469,-1.581,-47.503,179.747,6.112,149.175
C00625=1153.474,-1.830,-47.490,179.744,6.110,149.176
C00626=1153.479,-2.080,-47.476,179.742,6.110,149.176
C00627=1153.484,-2.329,-47.464,179.739,6.109,149.177
C00628=1153.489,-2.580,-47.450,179.737,6.108,149.177
C00629=1153.494,-2.828,-47.437,179.734,6.108,149.178
C00630=1153.500,-3.078,-47.424,179.732,6.107,149.178
C00631=1153.505,-3.328,-47.411,179.729,6.107,149.179
C00632=1153.511,-3.578,-47.397,179.727,6.106,149.180
C00633=1153.515,-3.828,-47.385,179.724,6.105,149.180
C00634=1153.520,-4.076,-47.371,179.722,6.104,149.181
C00635=1153.526,-4.326,-47.358,179.719,6.103,149.181
C00636=1153.530,-4.576,-47.345,179.717,6.103,149.182
C00637=1153.536,-4.826,-47.332,179.714,6.102,149.183
C00638=1153.541,-5.075,-47.319,179.712,6.101,149.183
C00639=1153.546,-5.325,-47.306,179.709,6.101,149.184
C00640=1153.552,-5.575,-47.293,179.707,6.100,149.184
C00641=1153.556,-5.824,-47.279,179.704,6.100,149.185
C00642=1153.561,-6.073,-47.267,179.702,6.099,149.185
C00643=1153.567,-6.323,-47.254,179.700,6.098,149.186
C00644=1153.571,-6.573,-47.241,179.697,6.097,149.186
C00645=1153.577,-6.823,-47.227,179.694,6.096,149.187
C00646=1153.582,-7.072,-47.215,179.692,6.096,149.188
C00647=1153.587,-7.322,-47.202,179.689,6.095,149.188
C00648=1153.593,-7.572,-47.189,179.687,6.094,149.189
C00649=1153.598,-7.821,-47.176,179.685,6.094,149.189
C00650=1153.602,-8.071,-47.163,179.682,6.093,149.190
C00651=1153.608,-8.320,-47.151,179.680,6.093,149.191
C00652=1153.613,-8.570,-47.137,179.678,6.092,149.191
C00653=1153.618,-8.820,-47.124,179.675,6.091,149.192
C00654=1153.623,-9.069,-47.111,179.673,6.091,149.192
C00655=1153.629,-9.318,-47.098,179.670,6.090,149.193
C00656=1153.634,-9.568,-47.085,179.667,6.089,149.193
C00657=1153.638,-9.818,-47.072,179.665,6.088,149.194
C00658=1153.643,-10.067,-47.060,179.662,6.087,149.195
C00659=1153.650,-10.317,-47.047,179.660,6.087,149.195
C00660=1153.654,-10.567,-47.034,179.658,6.086,149.196
C00661=1153.659,-10.816,-47.022,179.655,6.086,149.196
C00662=1153.664,-11.066,-47.009,179.653,6.085,149.197
C00663=1153.670,-11.315,-46.996,179.650,6.084,149.198
C00664=1153.675,-11.565,-46.983,179.648,6.084,149.198
C00665=1153.680,-11.815,-46.970,179.645,6.083,149.199
C00666=1153.685,-12.064,-46.958,179.643,6.082,149.199
C00667=1153.690,-12.314,-46.944,179.641,6.081,149.200
C00668=1153.695,-12.564,-46.932,179.638,6.081,149.200
C00669=1153.700,-12.813,-46.919,179.636,6.080,149.201
C00670=1153.706,-13.062,-46.906,179.633,6.080,149.202
C00671=1153.710,-13.312,-46.893,179.631,6.079,149.202
C00672=1153.716,-13.563,-46.881,179.629,6.079,149.203
C00673=1153.721,-13.812,-46.868,179.626,6.077,149.203
C00674=1153.726,-14.061,-46.856,179.623,6.077,149.204
C00675=1153.732,-14.311,-46.843,179.621,6.076,149.204
C00676=1153.736,-14.561,-46.830,179.618,6.075,149.205
C00677=1153.741,-14.810,-46.817,179.616,6.074,149.205
C00678=1153.747,-15.060,-46.805,179.613,6.074,149.206
C00679=1153.753,-15.309,-46.792,179.611,6.073,149.207
C00680=1153.757,-15.560,-46.779,179.609,6.073,149.207
C00681=1153.762,-15.809,-46.767,179.606,6.072,149.208
C00682=1153.767,-16.058,-46.754,179.604,6.072,149.209
C00683=1153.773,-16.308,-46.742,179.602,6.071,149.209
C00684=1153.778,-16.557,-46.730,179.599,6.070,149.210
C00685=1153.782,-16.807,-46.717,179.597,6.070,149.210
C00686=1153.788,-17.057,-46.704,179.594,6.069,149.211
C00687=1153.794,-17.307,-46.692,179.592,6.068,149.211
C00688=1153.799,-17.556,-46.679,179.589,6.068,149.212
C00689=1153.804,-17.806,-46.667,179.587,6.067,149.212
C00690=1153.809,-18.055,-46.654,179.584,6.067,149.213
C00691=1153.814,-18.306,-46.642,179.582,6.066,149.214
C00692=1153.819,-18.555,-46.629,179.580,6.065,149.214
C00693=1153.824,-18.804,-46.616,179.577,6.065,149.215
C00694=1153.830,-19.054,-46.605,179.575,6.064,149.215
C00695=1153.835,-19.303,-46.592,179.573,6.063,149.216
C00696=1153.840,-19.553,-46.579,179.570,6.063,149.217
C00697=1153.845,-19.803,-46.567,179.568,6.062,149.217
C00698=1153.850,-20.053,-46.555,179.565,6.062,149.218
C00699=1153.855,-20.302,-46.542,179.563,6.061,149.218
C00700=1153.860,-20.552,-46.530,179.560,6.060,149.219
C00701=1153.866,-20.802,-46.517,179.558,6.060,149.219
C00702=1153.871,-21.051,-46.504,179.555,6.059,149.220
C00703=1153.877,-21.301,-46.492,179.553,6.058,149.221
C00704=1153.882,-21.550,-46.480,179.551,6.058,149.221
C00705=1153.887,-21.800,-46.468,179.548,6.057,149.222
C00706=1153.892,-22.049,-46.455,179.546,6.057,149.222
C00707=1153.897,-22.299,-46.442,179.544,6.056,149.223
C00708=1153.902,-22.549,-46.430,179.541,6.056,149.224
C00709=1153.907,-22.799,-46.418,179.539,6.055,149.224
C00710=1153.912,-23.048,-46.407,179.536,6.054,149.225
C00711=1153.917,-23.298,-46.394,179.534,6.054,149.225
C00712=1153.923,-23.548,-46.382,179.531,6.053,149.226
C00713=1153.928,-23.797,-46.369,179.529,6.052,149.226
C00714=1153.934,-24.068,-46.356,179.526,6.052,149.227
C00715=1153.939,-24.337,-46.343,179.524,6.050,149.228
C00716=1153.945,-24.607,-46.330,179.521,6.050,149.228
C00717=1153.950,-24.877,-46.317,179.518,6.049,149.229
C00718=1153.955,-25.127,-46.304,179.516,6.049,149.229
C00719=1153.961,-25.377,-46.292,179.513,6.048,149.230
C00720=1153.966,-25.626,-46.280,179.511,6.047,149.231
C00721=1153.971,-25.876,-46.268,179.509,6.047,149.231
C00722=1153.976,-26.125,-46.255,179.506,6.046,149.232
C00723=1153.982,-26.375,-46.243,179.504,6.046,149.233
C00724=1153.987,-26.624,-46.231,179.502,6.045,149.233
C00725=1153.992,-26.874,-46.219,179.499,6.045,149.234
C00726=1153.997,-27.123,-46.207,179.497,6.044,149.234
C00727=1154.002,-27.373,-46.195,179.494,6.043,149.235
C00728=1154.008,-27.623,-46.183,179.492,6.043,149.235
C00729=1154.013,-27.873,-46.170,179.489,6.042,149.236
C00730=1154.018,-28.122,-46.158,179.487,6.041,149.237
C00731=1154.023,-28.372,-46.146,179.485,6.042,149.237
C00732=1154.029,-28.622,-46.134,179.483,6.041,149.238
C00733=1154.033,-28.871,-46.123,179.480,6.040,149.238
C00734=1154.038,-29.121,-46.110,179.478,6.040,149.239
C00735=1154.044,-29.371,-46.098,179.476,6.039,149.239
C00736=1154.049,-29.621,-46.086,179.473,6.038,149.240
C00737=1154.054,-29.870,-46.074,179.471,6.038,149.240
C00738=1154.059,-30.119,-46.062,179.468,6.037,149.241
C00739=1154.065,-30.369,-46.050,179.466,6.036,149.242
C00740=1154.070,-30.619,-46.038,179.463,6.036,149.242
C00741=1154.075,-30.869,-46.026,179.461,6.035,149.243
C00742=1154.081,-31.119,-46.014,179.459,6.035,149.244
C00743=1154.085,-31.368,-46.002,179.456,6.034,149.244
C00744=1154.090,-31.618,-45.990,179.454,6.034,149.245
C00745=1154.096,-31.867,-45.978,179.451,6.033,149.245
C00746=1154.101,-32.117,-45.966,179.449,6.032,149.246
C00747=1154.106,-32.366,-45.954,179.447,6.032,149.246
C00748=1154.111,-32.616,-45.943,179.444,6.031,149.247
C00749=1154.116,-32.866,-45.931,179.442,6.030,149.248
C00750=1154.122,-33.116,-45.918,179.439,6.030,149.248
C00751=1154.127,-33.365,-45.907,179.438,6.030,149.249
C00752=1154.132,-33.614,-45.895,179.435,6.030,149.249
C00753=1154.138,-33.864,-45.883,179.433,6.029,149.250
C00754=1154.143,-34.114,-45.872,179.430,6.028,149.251
C00755=1154.148,-34.363,-45.860,179.428,6.027,149.251
C00756=1154.153,-34.613,-45.848,179.425,6.027,149.252
C00757=1154.158,-34.863,-45.836,179.423,6.026,149.252
C00758=1154.163,-35.113,-45.824,179.421,6.025,149.253
C00759=1154.169,-35.363,-45.813,179.418,6.025,149.253
C00760=1154.174,-35.613,-45.801,179.416,6.024,149.254
C00761=1154.178,-35.862,-45.789,179.413,6.024,149.255
C00762=1154.184,-36.111,-45.777,179.411,6.023,149.255
C00763=1154.190,-36.361,-45.765,179.408,6.023,149.256
C00764=1154.195,-36.611,-45.753,179.406,6.022,149.256
C00765=1154.200,-36.860,-45.742,179.404,6.022,149.257
C00766=1154.205,-37.110,-45.730,179.402,6.021,149.257
C00767=1154.210,-37.360,-45.719,179.399,6.021,149.258
C00768=1154.216,-37.610,-45.707,179.397,6.020,149.259
C00769=1154.221,-37.859,-45.694,179.395,6.020,149.259
C00770=1154.226,-38.108,-45.684,179.392,6.019,149.260
C00771=1154.231,-38.358,-45.672,179.390,6.019,149.260
C00772=1154.237,-38.608,-45.660,179.387,6.018,149.261
C00773=1154.241,-38.858,-45.648,179.385,6.017,149.262
C00774=1154.247,-39.108,-45.637,179.383,6.017,149.262
C00775=1154.252,-39.358,-45.625,179.380,6.016,149.263
C00776=1154.258,-39.606,-45.614,179.378,6.016,149.263
C00777=1154.263,-39.856,-45.602,179.376,6.015,149.264
C00778=1154.268,-40.106,-45.591,179.374,6.015,149.264
C00779=1154.273,-40.356,-45.579,179.371,6.014,149.265
C00780=1154.278,-40.606,-45.567,179.369,6.014,149.266
C00781=1154.283,-40.856,-45.556,179.366,6.013,149.266
C00782=1154.289,-41.105,-45.544,179.364,6.013,149.267
C00783=1154.294,-41.354,-45.533,179.362,6.012,149.267
C00784=1154.299,-41.604,-45.521,179.359,6.011,149.268
C00785=1154.304,-41.854,-45.510,179.357,6.011,149.268
C00786=1154.310,-42.104,-45.498,179.355,6.011,149.269
C00787=1154.315,-42.353,-45.487,179.353,6.010,149.270
C00788=1154.320,-42.603,-45.475,179.350,6.010,149.270
C00789=1154.325,-42.852,-45.464,179.348,6.009,149.271
C00790=1154.330,-43.102,-45.452,179.346,6.008,149.271
C00791=1154.335,-43.352,-45.440,179.343,6.008,149.272
C00792=1154.341,-43.602,-45.430,179.341,6.007,149.272
C00793=1154.346,-43.851,-45.418,179.338,6.007,149.273
C00794=1154.352,-44.101,-45.406,179.336,6.007,149.274
C00795=1154.356,-44.351,-45.395,179.334,6.006,149.274
C00796=1154.362,-44.600,-45.384,179.332,6.005,149.275
C00797=1154.367,-44.850,-45.372,179.329,6.005,149.275
C00798=1154.372,-45.100,-45.360,179.327,6.004,149.276
C00799=1154.377,-45.349,-45.349,179.324,6.004,149.277
C00800=1154.383,-45.599,-45.337,179.322,6.003,149.277
C00801=1154.388,-45.849,-45.327,179.320,6.002,149.278
C00802=1154.394,-46.099,-45.315,179.318,6.003,149.278
C00803=1154.398,-46.348,-45.304,179.315,6.002,149.279
C00804=1154.404,-46.598,-45.292,179.313,6.001,149.280
C00805=1154.409,-46.847,-45.281,179.311,6.001,149.280
C00806=1154.414,-47.098,-45.270,179.308,6.000,149.281
C00807=1154.419,-47.348,-45.259,179.306,5.999,149.281
C00808=1154.425,-47.596,-45.248,179.303,5.999,149.282
C00809=1154.430,-47.846,-45.236,179.301,5.999,149.282
C00810=1154.435,-48.096,-45.224,179.299,5.999,149.283
C00811=1154.441,-48.346,-45.214,179.297,5.998,149.284
C00812=1154.446,-48.595,-45.202,179.294,5.997,149.284
C00813=1154.451,-48.845,-45.191,179.292,5.997,149.285
C00814=1154.456,-49.095,-45.179,179.290,5.996,149.285
C00815=1154.462,-49.345,-45.169,179.287,5.995,149.286
C00816=1154.467,-49.595,-45.157,179.285,5.995,149.286
C00817=1154.472,-49.844,-45.146,179.283,5.995,149.287
C00818=1154.478,-50.114,-45.134,179.280,5.994,149.288
C00819=1154.484,-50.385,-45.122,179.278,5.994,149.288
C00820=1154.488,-50.656,-45.110,179.275,5.993,149.289
C00821=1154.495,-50.926,-45.098,179.273,5.993,149.289
C00822=1154.500,-51.176,-45.086,179.270,5.992,149.290
C00823=1154.505,-51.426,-45.075,179.268,5.991,149.291
C00824=1154.510,-51.675,-45.065,179.265,5.991,149.291
C00825=1154.516,-51.925,-45.053,179.263,5.990,149.292
C00826=1154.521,-52.174,-45.042,179.261,5.991,149.292
C00827=1154.526,-52.425,-45.031,179.259,5.990,149.293
C00828=1154.531,-52.675,-45.019,179.257,5.989,149.293
C00829=1154.537,-52.923,-45.009,179.254,5.989,149.294
C00830=1154.542,-53.174,-44.998,179.252,5.988,149.295
C00831=1154.546,-53.423,-44.987,179.249,5.988,149.295
C00832=1154.553,-53.673,-44.976,179.248,5.988,149.296
C00833=1154.557,-53.923,-44.965,179.245,5.987,149.297
C00834=1154.562,-54.172,-44.953,179.243,5.986,149.297
C00835=1154.569,-54.422,-44.943,179.240,5.986,149.298
C00836=1154.573,-54.672,-44.931,179.238,5.985,149.298
C00837=1154.579,-54.921,-44.921,179.236,5.984,149.299
C00838=1154.584,-55.171,-44.910,179.234,5.985,149.299
C00839=1154.589,-55.421,-44.898,179.231,5.984,149.300
C00840=1154.595,-55.671,-44.888,179.229,5.984,149.301
C00841=1154.599,-55.920,-44.876,179.227,5.983,149.301
C00842=1154.604,-56.170,-44.866,179.224,5.982,149.302
C00843=1154.610,-56.419,-44.855,179.222,5.982,149.302
C00844=1154.615,-56.670,-44.844,179.220,5.982,149.303
C00845=1154.621,-56.919,-44.833,179.218,5.981,149.303
C00846=1154.626,-57.169,-44.822,179.215,5.980,149.304
C00847=1154.630,-57.419,-44.811,179.213,5.980,149.305
C00848=1154.637,-57.669,-44.800,179.211,5.980,149.305
C00849=1154.641,-57.918,-44.789,179.208,5.980,149.306
C00850=1154.647,-58.168,-44.779,179.206,5.979,149.306
C00851=1154.652,-58.417,-44.767,179.204,5.978,149.307
C00852=1154.657,-58.667,-44.757,179.201,5.978,149.307
C00853=1154.662,-58.916,-44.746,179.199,5.977,149.308
C00854=1154.668,-59.167,-44.735,179.197,5.977,149.309
C00855=1154.673,-59.416,-44.724,179.195,5.976,149.309
C00856=1154.678,-59.666,-44.713,179.192,5.976,149.310
C00857=1154.683,-59.916,-44.703,179.190,5.975,149.310
C00858=1154.688,-60.165,-44.692,179.188,5.976,149.311
C00859=1154.694,-60.415,-44.681,179.186,5.975,149.311
C00860=1154.698,-60.665,-44.670,179.184,5.974,149.312
C00861=1154.705,-60.914,-44.659,179.181,5.974,149.313
C00862=1154.710,-61.165,-44.649,179.179,5.973,149.313
C00863=1154.715,-61.414,-44.638,179.177,5.973,149.314
C00864=1154.720,-61.664,-44.627,179.174,5.973,149.314
C00865=1154.725,-61.913,-44.616,179.172,5.972,149.315
C00866=1154.730,-62.163,-44.606,179.170,5.971,149.315
C00867=1154.736,-62.413,-44.596,179.167,5.971,149.316
C00868=1154.741,-62.662,-44.584,179.165,5.971,149.317
C00869=1154.746,-62.912,-44.574,179.163,5.970,149.317
C00870=1154.752,-63.162,-44.563,179.160,5.970,149.318
C00871=1154.757,-63.411,-44.552,179.158,5.969,149.318
C00872=1154.762,-63.661,-44.541,179.157,5.969,149.319
C00873=1154.768,-63.911,-44.531,179.154,5.969,149.320
C00874=1154.773,-64.161,-44.521,179.152,5.968,149.320
C00875=1154.778,-64.410,-44.510,179.149,5.968,149.321
C00876=1154.783,-64.660,-44.499,179.147,5.967,149.321
C00877=1154.789,-64.910,-44.489,179.145,5.967,149.322
C00878=1154.793,-65.160,-44.478,179.143,5.966,149.322
C00879=1154.799,-65.409,-44.467,179.141,5.966,149.323
C00880=1154.804,-65.659,-44.457,179.138,5.965,149.324
C00881=1154.810,-65.909,-44.447,179.136,5.965,149.324
C00882=1154.814,-66.159,-44.435,179.134,5.965,149.325
C00883=1154.820,-66.408,-44.425,179.131,5.964,149.325
C00884=1154.825,-66.658,-44.415,179.129,5.963,149.326
C00885=1154.831,-66.908,-44.404,179.127,5.964,149.326
C00886=1154.836,-67.157,-44.393,179.125,5.963,149.327
C00887=1154.841,-67.407,-44.383,179.122,5.962,149.328
C00888=1154.846,-67.657,-44.373,179.120,5.962,149.328
C00889=1154.851,-67.907,-44.362,179.119,5.962,149.329
C00890=1154.857,-68.156,-44.352,179.116,5.961,149.329
C00891=1154.862,-68.407,-44.341,179.114,5.961,149.330
C00892=1154.867,-68.656,-44.330,179.111,5.960,149.330
C00893=1154.873,-68.905,-44.320,179.109,5.960,149.331
C00894=1154.878,-69.155,-44.310,179.107,5.959,149.331
C00895=1154.884,-69.405,-44.299,179.105,5.959,149.332
C00896=1154.889,-69.655,-44.289,179.102,5.958,149.333
C00897=1154.894,-69.905,-44.279,179.100,5.959,149.333
C00898=1154.899,-70.154,-44.268,179.098,5.958,149.334
C00899=1154.904,-70.404,-44.257,179.096,5.957,149.334
C00900=1154.910,-70.653,-44.247,179.093,5.957,149.335
C00901=1154.915,-70.904,-44.236,179.092,5.957,149.335
C00902=1154.921,-71.153,-44.226,179.089,5.956,149.336
C00903=1154.926,-71.403,-44.216,179.087,5.956,149.337
C00904=1154.931,-71.653,-44.205,179.085,5.955,149.337
C00905=1154.936,-71.902,-44.196,179.083,5.955,149.338
C00906=1154.942,-72.152,-44.185,179.080,5.954,149.338
C00907=1154.947,-72.402,-44.175,179.078,5.954,149.339
C00908=1154.952,-72.651,-44.165,179.075,5.953,149.339
C00909=1154.957,-72.902,-44.154,179.074,5.953,149.340
C00910=1154.963,-73.151,-44.144,179.071,5.953,149.341
C00911=1154.968,-73.400,-44.133,179.069,5.952,149.341
C00912=1154.973,-73.650,-44.122,179.067,5.952,149.342
C00913=1154.979,-73.900,-44.112,179.065,5.952,149.342
C00914=1154.984,-74.150,-44.102,179.063,5.951,149.343
C00915=1154.989,-74.399,-44.092,179.060,5.951,149.344
C00916=1154.994,-74.649,-44.082,179.058,5.951,149.344
C00917=1155.000,-74.899,-44.072,179.056,5.950,149.345
C00918=1155.005,-75.149,-44.061,179.053,5.949,149.345
C00919=1155.010,-75.398,-44.051,179.051,5.949,149.346
C00920=1155.016,-75.648,-44.041,179.049,5.949,149.346
C00921=1155.021,-75.898,-44.031,179.047,5.948,149.347
C00922=1155.027,-76.169,-44.020,179.044,5.948,149.348
C00923=1155.032,-76.441,-44.009,179.042,5.947,149.348
C00924=1155.038,-76.712,-43.998,179.039,5.947,149.349
C00925=1155.044,-76.983,-43.987,179.038,5.947,149.349
C00926=1155.049,-77.233,-43.977,179.035,5.946,149.350
C00927=1155.055,-77.483,-43.966,179.033,5.946,149.350
C00928=1155.060,-77.732,-43.956,179.031,5.945,149.351
C00929=1155.066,-77.982,-43.946,179.029,5.945,149.352
C00930=1155.070,-78.232,-43.936,179.027,5.944,149.352
C00931=1155.076,-78.482,-43.926,179.024,5.944,149.353
C00932=1155.082,-78.731,-43.916,179.022,5.944,149.353
C00933=1155.087,-78.981,-43.906,179.020,5.943,149.354
C00934=1155.092,-79.231,-43.895,179.017,5.943,149.355
C00935=1155.097,-79.480,-43.886,179.016,5.943,149.355
C00936=1155.103,-79.730,-43.876,179.014,5.942,149.355
C00937=1155.108,-79.980,-43.865,179.011,5.942,149.356
C00938=1155.113,-80.230,-43.855,179.009,5.941,149.357
C00939=1155.118,-80.480,-43.846,179.007,5.941,149.357
C00940=1155.124,-80.729,-43.836,179.004,5.941,149.358
C00941=1155.129,-80.979,-43.825,179.002,5.940,149.358
C00942=1155.134,-81.229,-43.816,179.000,5.940,149.359
C00943=1155.139,-81.478,-43.805,178.998,5.940,149.360
C00944=1155.145,-81.728,-43.796,178.996,5.939,149.360
C00945=1155.150,-81.979,-43.785,178.994,5.939,149.361
C00946=1155.155,-82.228,-43.776,178.992,5.938,149.361
C00947=1155.161,-82.477,-43.765,178.989,5.938,149.362
C00948=1155.166,-82.727,-43.755,178.987,5.938,149.362
C00949=1155.172,-82.977,-43.746,178.985,5.937,149.363
C00950=1155.177,-83.227,-43.736,178.983,5.936,149.363
C00951=1155.182,-83.476,-43.726,178.981,5.937,149.364
C00952=1155.187,-83.726,-43.716,178.979,5.936,149.365
C00953=1155.193,-83.976,-43.706,178.976,5.935,149.365
C00954=1155.198,-84.226,-43.696,178.974,5.935,149.366
C00955=1155.203,-84.475,-43.686,178.972,5.935,149.366
C00956=1155.208,-84.725,-43.676,178.969,5.935,149.367
C00957=1155.214,-84.975,-43.667,178.967,5.934,149.367
C00958=1155.219,-85.224,-43.657,178.966,5.934,149.368
C00959=1155.224,-85.475,-43.646,178.963,5.933,149.369
C00960=1155.229,-85.724,-43.637,178.961,5.933,149.369
C00961=1155.235,-85.974,-43.627,178.959,5.933,149.370
C00962=1155.240,-86.223,-43.617,178.957,5.932,149.370
C00963=1155.246,-86.473,-43.608,178.954,5.932,149.371
C00964=1155.251,-86.723,-43.598,178.953,5.932,149.371
C00965=1155.256,-86.973,-43.587,178.950,5.931,149.372
C00966=1155.261,-87.223,-43.578,178.948,5.930,149.372
C00967=1155.267,-87.472,-43.568,178.946,5.930,149.373
C00968=1155.272,-87.722,-43.559,178.944,5.930,149.374
C00969=1155.278,-87.972,-43.549,178.941,5.929,149.374
C00970=1155.283,-88.221,-43.540,178.940,5.929,149.375
C00971=1155.288,-88.471,-43.529,178.937,5.929,149.375
C00972=1155.294,-88.722,-43.519,178.935,5.928,149.376
C00973=1155.298,-88.971,-43.510,178.933,5.928,149.376
C00974=1155.304,-89.221,-43.500,178.931,5.928,149.377
C00975=1155.309,-89.470,-43.491,178.929,5.928,149.377
C00976=1155.315,-89.720,-43.481,178.927,5.927,149.378
C00977=1155.320,-89.970,-43.472,178.924,5.927,149.379
C00978=1155.325,-90.220,-43.461,178.923,5.927,149.379
C00979=1155.330,-90.470,-43.452,178.920,5.926,149.380
C00980=1155.336,-90.719,-43.442,178.918,5.926,149.380
C00981=1155.341,-90.969,-43.433,178.916,5.926,149.381
C00982=1155.346,-91.219,-43.423,178.914,5.925,149.381
C00983=1155.352,-91.469,-43.413,178.911,5.924,149.382
C00984=1155.357,-91.718,-43.404,178.910,5.925,149.383
C00985=1155.363,-91.968,-43.394,178.908,5.924,149.383
C00986=1155.368,-92.217,-43.385,178.905,5.923,149.384
C00987=1155.373,-92.468,-43.375,178.903,5.923,149.384
C00988=1155.378,-92.717,-43.365,178.901,5.923,149.385
C00989=1155.384,-92.968,-43.356,178.899,5.922,149.385
C00990=1155.389,-93.217,-43.346,178.897,5.922,149.386
C00991=1155.394,-93.467,-43.337,178.895,5.922,149.386
C00992=1155.400,-93.716,-43.327,178.893,5.922,149.387
C00993=1155.405,-93.966,-43.318,178.890,5.921,149.388
C00994=1155.410,-94.216,-43.308,178.888,5.920,149.388
C00995=1155.416,-94.466,-43.299,178.887,5.920,149.389
C00996=1155.421,-94.715,-43.289,178.884,5.920,149.389
C00997=1155.426,-94.965,-43.280,178.882,5.919,149.390
C00998=1155.432,-95.214,-43.270,178.880,5.919,149.390
C00999=1155.437,-95.464,-43.261,178.877,5.919,149.391
C01000=1155.443,-95.714,-43.251,178.876,5.919,149.391
C01001=1155.447,-95.964,-43.241,178.874,5.918,149.392
C01002=1155.452,-96.214,-43.232,178.871,5.918,149.393
C01003=1155.458,-96.464,-43.222,178.869,5.918,149.393
C01004=1155.463,-96.714,-43.213,178.867,5.917,149.394
C01005=1155.469,-96.964,-43.204,178.865,5.916,149.394
C01006=1155.474,-97.213,-43.194,178.863,5.917,149.395
C01007=1155.480,-97.463,-43.185,178.861,5.916,149.395
C01008=1155.485,-97.712,-43.175,178.859,5.916,149.396
C01009=1155.490,-97.962,-43.166,178.856,5.916,149.396
C01010=1155.496,-98.212,-43.157,178.854,5.915,149.397
C01011=1155.501,-98.462,-43.147,178.853,5.915,149.397
C01012=1155.506,-98.712,-43.138,178.850,5.914,149.398
C01013=1155.512,-98.962,-43.129,178.848,5.915,149.399
C01014=1155.517,-99.211,-43.119,178.846,5.914,149.399
C01015=1155.522,-99.461,-43.110,178.844,5.913,149.400
C01016=1155.528,-99.711,-43.101,178.842,5.913,149.400
C01017=1155.533,-99.961,-43.092,178.840,5.913,149.401
C01018=1155.538,-100.210,-43.082,178.838,5.913,149.401
C01019=1155.544,-100.460,-43.073,178.835,5.912,149.402
C01020=1155.549,-100.710,-43.064,178.833,5.912,149.402
C01021=1155.554,-100.960,-43.054,178.832,5.912,149.403
C01022=1155.560,-101.209,-43.045,178.829,5.911,149.403
C01023=1155.565,-101.459,-43.036,178.827,5.910,149.404
C01024=1155.571,-101.709,-43.026,178.825,5.911,149.405
C01025=1155.575,-101.959,-43.017,178.823,5.910,149.405
C01026=1155.582,-102.231,-43.008,178.821,5.910,149.406
C01027=1155.587,-102.502,-42.997,178.819,5.909,149.406
C01028=1155.593,-102.774,-42.987,178.816,5.909,149.407
C01029=1155.599,-103.047,-42.976,178.814,5.908,149.408
C01030=1155.604,-103.296,-42.967,178.812,5.908,149.408
C01031=1155.609,-103.546,-42.958,178.810,5.908,149.409
C01032=1155.615,-103.796,-42.950,178.808,5.908,149.409
C01033=1155.620,-104.046,-42.940,178.806,5.907,149.410
C01034=1155.625,-104.296,-42.930,178.804,5.906,149.410
C01035=1155.631,-104.545,-42.922,178.802,5.907,149.411
C01036=1155.636,-104.795,-42.913,178.799,5.906,149.411
C01037=1155.642,-105.045,-42.903,178.798,5.906,149.412
C01038=1155.647,-105.295,-42.895,178.795,5.906,149.413
C01039=1155.653,-105.544,-42.886,178.793,5.905,149.413
C01040=1155.657,-105.794,-42.876,178.791,5.905,149.414
C01041=1155.663,-106.044,-42.867,178.789,5.904,149.414
C01042=1155.668,-106.294,-42.858,178.787,5.905,149.415
C01043=1155.674,-106.544,-42.849,178.785,5.904,149.415
C01044=1155.679,-106.793,-42.840,178.783,5.904,149.416
C01045=1155.684,-107.043,-42.831,178.781,5.903,149.416
C01046=1155.690,-107.293,-42.822,178.778,5.903,149.417
C01047=1155.695,-107.543,-42.812,178.777,5.903,149.417
C01048=1155.700,-107.792,-42.803,178.775,5.902,149.418
C01049=1155.706,-108.042,-42.794,178.773,5.902,149.418
C01050=1155.711,-108.291,-42.786,178.770,5.902,149.419
C01051=1155.717,-108.542,-42.776,178.769,5.902,149.420
C01052=1155.722,-108.791,-42.767,178.766,5.901,149.420
C01053=1155.727,-109.041,-42.758,178.764,5.900,149.421
C01054=1155.732,-109.291,-42.749,178.762,5.901,149.421
C01055=1155.737,-109.541,-42.740,178.760,5.900,149.422
C01056=1155.743,-109.791,-42.731,178.758,5.900,149.422
C01057=1155.749,-110.040,-42.722,178.756,5.899,149.423
C01058=1155.754,-110.290,-42.714,178.754,5.900,149.423
C01059=1155.759,-110.540,-42.705,178.752,5.899,149.424
C01060=1155.765,-110.790,-42.696,178.750,5.898,149.424
C01061=1155.770,-111.040,-42.687,178.748,5.898,149.425
C01062=1155.775,-111.290,-42.678,178.746,5.897,149.425
C01063=1155.781,-111.540,-42.668,178.744,5.898,149.426
C01064=1155.787,-111.789,-42.660,178.742,5.897,149.427
C01065=1155.792,-112.039,-42.651,178.740,5.897,149.427
C01066=1155.797,-112.289,-42.642,178.738,5.896,149.428
C01067=1155.802,-112.538,-42.633,178.736,5.897,149.428
C01068=1155.807,-112.788,-42.624,178.734,5.896,149.429
C01069=1155.812,-113.038,-42.615,178.731,5.895,149.429
C01070=1155.818,-113.287,-42.607,178.730,5.895,149.430
C01071=1155.824,-113.537,-42.597,178.727,5.895,149.430
C01072=1155.829,-113.787,-42.589,178.726,5.895,149.431
C01073=1155.834,-114.037,-42.580,178.723,5.894,149.431
C01074=1155.840,-114.287,-42.571,178.722,5.894,149.432
C01075=1155.845,-114.536,-42.562,178.720,5.893,149.432
C01076=1155.850,-114.786,-42.553,178.717,5.894,149.433
C01077=1155.856,-115.036,-42.544,178.715,5.893,149.434
C01078=1155.861,-115.286,-42.536,178.714,5.893,149.434
C01079=1155.866,-115.536,-42.527,178.711,5.892,149.435
C01080=1155.872,-115.785,-42.519,178.709,5.892,149.435
C01081=1155.877,-116.035,-42.510,178.707,5.892,149.436
C01082=1155.882,-116.285,-42.501,178.705,5.891,149.436
C01083=1155.888,-116.535,-42.492,178.703,5.891,149.437
C01084=1155.893,-116.785,-42.483,178.701,5.891,149.437
C01085=1155.898,-117.034,-42.475,178.700,5.891,149.438
C01086=1155.904,-117.284,-42.466,178.697,5.890,149.438
C01087=1155.909,-117.534,-42.457,178.695,5.890,149.439
C01088=1155.915,-117.784,-42.448,178.693,5.890,149.439
C01089=1155.921,-118.034,-42.440,178.692,5.890,149.440
C01090=1155.926,-118.283,-42.431,178.689,5.889,149.440
C01091=1155.931,-118.533,-42.422,178.687,5.889,149.441
C01092=1155.936,-118.783,-42.413,178.685,5.889,149.442
C01093=1155.942,-119.032,-42.404,178.683,5.889,149.442
C01094=1155.947,-119.282,-42.397,178.681,5.888,149.443
C01095=1155.952,-119.532,-42.388,178.679,5.887,149.443
C01096=1155.957,-119.782,-42.379,178.677,5.888,149.444
C01097=1155.963,-120.031,-42.370,178.675,5.887,149.444
C01098=1155.968,-120.281,-42.362,178.673,5.887,149.445
C01099=1155.974,-120.532,-42.353,178.671,5.886,149.445
C01100=1155.979,-120.781,-42.344,178.669,5.886,149.446
C01101=1155.984,-121.031,-42.336,178.667,5.886,149.446
C01102=1155.990,-121.280,-42.327,178.665,5.886,149.447
C01103=1155.995,-121.531,-42.319,178.663,5.885,149.447
C01104=1156.000,-121.781,-42.310,178.661,5.885,149.448
C01105=1156.006,-122.030,-42.301,178.659,5.884,149.448
C01106=1156.011,-122.280,-42.293,178.658,5.884,149.449
C01107=1156.017,-122.530,-42.284,178.655,5.884,149.450
C01108=1156.022,-122.779,-42.276,178.653,5.884,149.450
C01109=1156.028,-123.029,-42.267,178.651,5.883,149.451
C01110=1156.033,-123.280,-42.259,178.649,5.883,149.451
C01111=1156.038,-123.530,-42.250,178.647,5.883,149.452
C01112=1156.043,-123.778,-42.242,178.645,5.883,149.452
C01113=1156.049,-124.029,-42.234,178.643,5.882,149.453
C01114=1156.054,-124.279,-42.225,178.641,5.882,149.453
C01115=1156.060,-124.528,-42.216,178.639,5.881,149.454
C01116=1156.065,-124.778,-42.207,178.638,5.882,149.454
C01117=1156.070,-125.028,-42.199,178.635,5.881,149.455
C01118=1156.076,-125.277,-42.191,178.634,5.881,149.455
C01119=1156.081,-125.527,-42.182,178.631,5.880,149.456
C01120=1156.087,-125.778,-42.174,178.630,5.880,149.456
C01121=1156.092,-126.026,-42.166,178.627,5.880,149.457
C01122=1156.097,-126.277,-42.157,178.626,5.880,149.457
C01123=1156.102,-126.527,-42.149,178.624,5.879,149.458
C01124=1156.108,-126.776,-42.140,178.622,5.879,149.458
C01125=1156.114,-127.026,-42.132,178.619,5.879,149.459
C01126=1156.119,-127.276,-42.123,178.618,5.879,149.460
C01127=1156.125,-127.526,-42.115,178.615,5.878,149.460
C01128=1156.129,-127.776,-42.107,178.614,5.878,149.460
C01129=1156.134,-128.025,-42.098,178.612,5.877,149.461
C01130=1155.714,-128.036,-42.141,178.608,5.881,149.463
C01131=1155.709,-127.787,-42.149,178.610,5.881,149.462
C01132=1155.703,-127.537,-42.157,178.612,5.882,149.462
C01133=1155.698,-127.287,-42.166,178.614,5.882,149.461
C01134=1155.692,-127.037,-42.174,178.617,5.882,149.461
C01135=1155.687,-126.787,-42.182,178.618,5.882,149.460
C01136=1155.682,-126.538,-42.191,178.620,5.883,149.460
C01137=1155.676,-126.288,-42.199,178.622,5.883,149.459
C01138=1155.671,-126.038,-42.207,178.624,5.884,149.459
C01139=1155.666,-125.788,-42.216,178.626,5.884,149.458
C01140=1155.660,-125.539,-42.224,178.628,5.884,149.457
C01141=1155.655,-125.289,-42.233,178.630,5.884,149.457
C01142=1155.649,-125.038,-42.241,178.632,5.885,149.456
C01143=1155.644,-124.789,-42.250,178.634,5.885,149.456
C01144=1155.638,-124.539,-42.259,178.636,5.886,149.456
C01145=1155.633,-124.289,-42.267,178.638,5.886,149.455
C01146=1155.628,-124.040,-42.275,178.640,5.886,149.455
C01147=1155.623,-123.790,-42.284,178.642,5.886,149.454
C01148=1155.617,-123.540,-42.292,178.644,5.887,149.453
C01149=1155.612,-123.291,-42.300,178.646,5.887,149.453
C01150=1155.606,-123.041,-42.309,178.648,5.887,149.452
C01151=1155.601,-122.791,-42.318,178.649,5.887,149.452
C01152=1155.596,-122.540,-42.326,178.652,5.888,149.451
C01153=1155.590,-122.291,-42.335,178.654,5.888,149.451
C01154=1155.585,-122.041,-42.344,178.656,5.888,149.450
C01155=1155.579,-121.791,-42.352,178.657,5.888,149.450
C01156=1155.574,-121.542,-42.361,178.660,5.889,149.449
C01157=1155.568,-121.292,-42.369,178.661,5.889,149.449
C01158=1155.564,-121.042,-42.378,178.663,5.890,149.448
C01159=1155.558,-120.792,-42.386,178.666,5.889,149.448
C01160=1155.553,-120.543,-42.394,178.668,5.890,149.447
C01161=1155.548,-120.293,-42.403,178.669,5.890,149.447
C01162=1155.542,-120.043,-42.412,178.672,5.891,149.446
C01163=1155.537,-119.794,-42.421,178.673,5.891,149.446
C01164=1155.531,-119.543,-42.429,178.676,5.891,149.445
C01165=1155.526,-119.294,-42.438,178.677,5.891,149.444
C01166=1155.521,-119.044,-42.447,178.680,5.892,149.444
C01167=1155.515,-118.795,-42.455,178.681,5.892,149.443
C01168=1155.510,-118.545,-42.464,178.683,5.893,149.443
C01169=1155.504,-118.294,-42.472,178.686,5.893,149.442
C01170=1155.499,-118.044,-42.481,178.688,5.893,149.442
C01171=1155.494,-117.795,-42.490,178.690,5.894,149.441
C01172=1155.488,-117.545,-42.499,178.691,5.894,149.441
C01173=1155.483,-117.296,-42.508,178.694,5.894,149.440
C01174=1155.478,-117.046,-42.517,178.696,5.894,149.440
C01175=1155.473,-116.795,-42.525,178.698,5.895,149.439
C01176=1155.467,-116.546,-42.533,178.700,5.895,149.439
C01177=1155.462,-116.296,-42.542,178.702,5.895,149.438
C01178=1155.456,-116.046,-42.551,178.703,5.895,149.438
C01179=1155.451,-115.797,-42.560,178.706,5.896,149.437
C01180=1155.445,-115.547,-42.569,178.708,5.896,149.436
C01181=1155.440,-115.297,-42.578,178.710,5.896,149.436
C01182=1155.434,-115.047,-42.587,178.711,5.896,149.435
C01183=1155.429,-114.798,-42.596,178.714,5.897,149.435
C01184=1155.424,-114.547,-42.604,178.716,5.898,149.434
C01185=1155.418,-114.298,-42.612,178.718,5.898,149.434
C01186=1155.413,-114.048,-42.621,178.720,5.898,149.433
C01187=1155.408,-113.798,-42.630,178.722,5.898,149.433
C01188=1155.403,-113.548,-42.639,178.724,5.899,149.432
C01189=1155.397,-113.299,-42.648,178.726,5.899,149.432
C01190=1155.392,-113.049,-42.657,178.728,5.899,149.431
C01191=1155.386,-112.800,-42.666,178.730,5.899,149.431
C01192=1155.381,-112.549,-42.675,178.732,5.900,149.430
C01193=1155.375,-112.299,-42.684,178.735,5.900,149.429
C01194=1155.370,-112.050,-42.693,178.736,5.900,149.429
C01195=1155.365,-111.800,-42.702,178.738,5.901,149.428
C01196=1155.360,-111.550,-42.711,178.740,5.901,149.428
C01197=1155.354,-111.301,-42.719,178.742,5.902,149.427
C01198=1155.349,-111.051,-42.728,178.744,5.901,149.427
C01199=1155.344,-110.801,-42.737,178.746,5.902,149.426
C01200=1155.338,-110.551,-42.746,178.748,5.902,149.426
C01201=1155.333,-110.301,-42.755,178.750,5.903,149.425
C01202=1155.328,-110.051,-42.764,178.753,5.903,149.425
C01203=1155.322,-109.801,-42.773,178.755,5.903,149.424
C01204=1155.317,-109.552,-42.782,178.757,5.904,149.424
C01205=1155.311,-109.302,-42.791,178.758,5.904,149.423
C01206=1155.305,-109.052,-42.800,178.761,5.904,149.422
C01207=1155.300,-108.802,-42.809,178.763,5.904,149.422
C01208=1155.295,-108.552,-42.818,178.765,5.905,149.421
C01209=1155.290,-108.303,-42.827,178.767,5.906,149.421
C01210=1155.285,-108.053,-42.836,178.769,5.905,149.420
C01211=1155.280,-107.804,-42.845,178.771,5.906,149.420
C01212=1155.273,-107.554,-42.854,178.773,5.906,149.419
C01213=1155.268,-107.304,-42.863,178.775,5.907,149.419
C01214=1155.263,-107.054,-42.872,178.777,5.907,149.418
C01215=1155.258,-106.805,-42.881,178.779,5.907,149.418
C01216=1155.252,-106.554,-42.891,178.782,5.908,149.417
C01217=1155.247,-106.305,-42.899,178.783,5.908,149.417
C01218=1155.242,-106.055,-42.908,178.786,5.908,149.416
C01219=1155.237,-105.805,-42.918,178.787,5.908,149.415
C01220=1155.232,-105.556,-42.927,178.790,5.909,149.415
C01221=1155.226,-105.305,-42.936,178.791,5.909,149.414
C01222=1155.221,-105.056,-42.945,178.794,5.909,149.414
C01223=1155.215,-104.806,-42.954,178.796,5.910,149.413
C01224=1155.210,-104.557,-42.963,178.798,5.910,149.413
C01225=1155.204,-104.307,-42.973,178.800,5.911,149.412
C01226=1155.199,-104.057,-42.982,178.802,5.910,149.412
C01227=1155.194,-103.807,-42.991,178.804,5.911,149.411
C01228=1155.189,-103.557,-43.000,178.806,5.912,149.411
C01229=1155.183,-103.307,-43.009,178.808,5.912,149.410
C01230=1155.178,-103.058,-43.019,178.811,5.912,149.409
C01231=1155.172,-102.786,-43.028,178.813,5.913,149.409
C01232=1155.167,-102.514,-43.038,178.815,5.913,149.408
C01233=1155.161,-102.242,-43.049,178.817,5.913,149.408
C01234=1155.154,-101.970,-43.058,178.820,5.914,149.407
C01235=1155.149,-101.720,-43.068,178.821,5.914,149.406
C01236=1155.144,-101.470,-43.077,178.824,5.914,149.406
C01237=1155.138,-101.220,-43.086,178.826,5.915,149.405
C01238=1155.133,-100.970,-43.095,178.828,5.915,149.405
C01239=1155.128,-100.721,-43.105,178.830,5.916,149.404
C01240=1155.123,-100.471,-43.114,178.832,5.916,149.404
C01241=1155.117,-100.221,-43.123,178.834,5.916,149.403
C01242=1155.112,-99.972,-43.133,178.836,5.917,149.403
C01243=1155.106,-99.722,-43.142,178.838,5.917,149.402
C01244=1155.101,-99.472,-43.151,178.840,5.917,149.402
C01245=1155.096,-99.223,-43.161,178.842,5.917,149.401
C01246=1155.090,-98.973,-43.170,178.845,5.918,149.400
C01247=1155.085,-98.723,-43.179,178.847,5.919,149.400
C01248=1155.080,-98.473,-43.189,178.848,5.919,149.399
C01249=1155.074,-98.223,-43.198,178.851,5.919,149.399
C01250=1155.069,-97.973,-43.207,178.853,5.919,149.398
C01251=1155.063,-97.724,-43.218,178.855,5.920,149.398
C01252=1155.058,-97.474,-43.226,178.857,5.920,149.397
C01253=1155.053,-97.224,-43.235,178.859,5.920,149.397
C01254=1155.048,-96.975,-43.246,178.861,5.921,149.396
C01255=1155.042,-96.725,-43.254,178.864,5.921,149.395
C01256=1155.036,-96.475,-43.264,178.866,5.921,149.395
C01257=1155.032,-96.225,-43.274,178.868,5.922,149.394
C01258=1155.026,-95.976,-43.282,178.869,5.922,149.394
C01259=1155.021,-95.725,-43.293,178.872,5.922,149.393
C01260=1155.016,-95.475,-43.302,178.874,5.923,149.393
C01261=1155.010,-95.225,-43.311,178.876,5.923,149.392
C01262=1155.006,-94.976,-43.321,178.878,5.923,149.392
C01263=1155.000,-94.726,-43.330,178.881,5.924,149.391
C01264=1154.995,-94.477,-43.340,178.882,5.924,149.391
C01265=1154.989,-94.227,-43.350,178.885,5.924,149.390
C01266=1154.984,-93.977,-43.359,178.886,5.924,149.389
C01267=1154.979,-93.727,-43.368,178.889,5.925,149.389
C01268=1154.973,-93.478,-43.378,178.891,5.926,149.388
C01269=1154.968,-93.228,-43.387,178.893,5.925,149.388
C01270=1154.962,-92.979,-43.397,178.895,5.926,149.387
C01271=1154.957,-92.729,-43.406,178.897,5.927,149.387
C01272=1154.952,-92.479,-43.417,178.899,5.927,149.386
C01273=1154.947,-92.229,-43.426,178.902,5.927,149.386
C01274=1154.942,-91.979,-43.436,178.904,5.928,149.385
C01275=1154.936,-91.729,-43.445,178.906,5.928,149.384
C01276=1154.931,-91.480,-43.455,178.908,5.928,149.384
C01277=1154.926,-91.230,-43.464,178.910,5.928,149.383
C01278=1154.920,-90.980,-43.474,178.912,5.929,149.383
C01279=1154.915,-90.730,-43.483,178.915,5.930,149.382
C01280=1154.909,-90.481,-43.493,178.916,5.930,149.382
C01281=1154.904,-90.231,-43.502,178.919,5.930,149.381
C01282=1154.898,-89.981,-43.512,178.921,5.931,149.381
C01283=1154.893,-89.731,-43.522,178.923,5.931,149.380
C01284=1154.888,-89.481,-43.532,178.925,5.931,149.379
C01285=1154.883,-89.232,-43.542,178.927,5.932,149.379
C01286=1154.878,-88.982,-43.551,178.929,5.932,149.378
C01287=1154.872,-88.732,-43.561,178.932,5.932,149.378
C01288=1154.867,-88.483,-43.570,178.934,5.933,149.377
C01289=1154.861,-88.233,-43.580,178.936,5.933,149.377
C01290=1154.857,-87.983,-43.590,178.938,5.933,149.376
C01291=1154.851,-87.733,-43.600,178.940,5.934,149.375
C01292=1154.845,-87.483,-43.610,178.942,5.934,149.375
C01293=1154.841,-87.234,-43.620,178.945,5.934,149.374
C01294=1154.835,-86.984,-43.629,178.947,5.935,149.374
C01295=1154.830,-86.735,-43.639,178.948,5.935,149.373
C01296=1154.825,-86.484,-43.649,178.951,5.936,149.373
C01297=1154.819,-86.234,-43.659,178.953,5.936,149.372
C01298=1154.814,-85.985,-43.668,178.955,5.936,149.372
C01299=1154.808,-85.735,-43.678,178.958,5.937,149.371
C01300=1154.803,-85.486,-43.688,178.960,5.937,149.370
C01301=1154.798,-85.235,-43.698,178.961,5.937,149.370
C01302=1154.793,-84.986,-43.708,178.964,5.938,149.369
C01303=1154.788,-84.736,-43.717,178.966,5.939,149.369
C01304=1154.782,-84.487,-43.727,178.968,5.939,149.368
C01305=1154.776,-84.237,-43.738,178.970,5.939,149.368
C01306=1154.772,-83.986,-43.747,178.973,5.940,149.367
C01307=1154.766,-83.737,-43.757,178.974,5.940,149.367
C01308=1154.761,-83.487,-43.767,178.977,5.940,149.366
C01309=1154.756,-83.238,-43.777,178.979,5.941,149.365
C01310=1154.750,-82.988,-43.786,178.981,5.941,149.365
C01311=1154.745,-82.738,-43.797,178.983,5.941,149.364
C01312=1154.740,-82.488,-43.807,178.986,5.942,149.364
C01313=1154.734,-82.239,-43.817,178.987,5.942,149.363
C01314=1154.729,-81.989,-43.827,178.990,5.942,149.363
C01315=1154.724,-81.739,-43.836,178.992,5.943,149.362
C01316=1154.719,-81.489,-43.846,178.994,5.943,149.362
C01317=1154.713,-81.240,-43.857,178.996,5.943,149.361
C01318=1154.707,-80.990,-43.867,178.999,5.944,149.360
C01319=1154.703,-80.741,-43.877,179.001,5.945,149.360
C01320=1154.697,-80.490,-43.886,179.003,5.945,149.359
C01321=1154.692,-80.241,-43.897,179.005,5.945,149.359
C01322=1154.687,-79.991,-43.906,179.008,5.946,149.358
C01323=1154.682,-79.741,-43.917,179.009,5.946,149.358
C01324=1154.676,-79.492,-43.927,179.011,5.947,149.357
C01325=1154.671,-79.242,-43.937,179.014,5.947,149.356
C01326=1154.665,-78.992,-43.946,179.016,5.947,149.356
C01327=1154.660,-78.742,-43.957,179.018,5.948,149.355
C01328=1154.655,-78.492,-43.967,179.021,5.948,149.355
C01329=1154.649,-78.243,-43.977,179.023,5.949,149.354
C01330=1154.644,-77.993,-43.987,179.025,5.948,149.353
C01331=1154.639,-77.743,-43.997,179.027,5.949,149.353
C01332=1154.634,-77.494,-44.007,179.029,5.950,149.353
C01333=1154.628,-77.244,-44.018,179.031,5.950,149.352
C01334=1154.623,-76.994,-44.028,179.033,5.950,149.351
C01335=1154.617,-76.723,-44.038,179.036,5.951,149.351
C01336=1154.611,-76.451,-44.050,179.038,5.951,149.350
C01337=1154.606,-76.180,-44.061,179.041,5.952,149.349
C01338=1154.599,-75.909,-44.072,179.043,5.953,149.349
C01339=1154.594,-75.659,-44.082,179.045,5.952,149.348
C01340=1154.590,-75.410,-44.092,179.047,5.953,149.348
C01341=1154.584,-75.160,-44.102,179.050,5.954,149.347
C01342=1154.579,-74.910,-44.113,179.052,5.953,149.347
C01343=1154.573,-74.660,-44.123,179.054,5.954,149.346
C01344=1154.568,-74.411,-44.133,179.057,5.955,149.345
C01345=1154.563,-74.160,-44.144,179.059,5.955,149.345
C01346=1154.557,-73.911,-44.154,179.060,5.955,149.344
C01347=1154.552,-73.662,-44.164,179.063,5.956,149.344
C01348=1154.547,-73.411,-44.174,179.065,5.956,149.343
C01349=1154.542,-73.162,-44.184,179.067,5.956,149.343
C01350=1154.536,-72.912,-44.195,179.070,5.957,149.342
C01351=1154.531,-72.662,-44.205,179.072,5.958,149.342
C01352=1154.526,-72.413,-44.215,179.074,5.958,149.341
C01353=1154.520,-72.163,-44.226,179.076,5.958,149.340
C01354=1154.515,-71.913,-44.236,179.078,5.959,149.340
C01355=1154.509,-71.663,-44.246,179.081,5.959,149.339
C01356=1154.504,-71.414,-44.257,179.083,5.960,149.339
C01357=1154.500,-71.164,-44.267,179.085,5.959,149.338
C01358=1154.494,-70.915,-44.277,179.087,5.960,149.338
C01359=1154.489,-70.665,-44.288,179.089,5.961,149.337
C01360=1154.484,-70.415,-44.298,179.092,5.961,149.336
C01361=1154.478,-70.165,-44.308,179.094,5.961,149.336
C01362=1154.473,-69.915,-44.319,179.096,5.962,149.335
C01363=1154.467,-69.666,-44.329,179.099,5.963,149.335
C01364=1154.462,-69.416,-44.339,179.101,5.963,149.334
C01365=1154.457,-69.166,-44.351,179.103,5.963,149.333
C01366=1154.451,-68.917,-44.361,179.105,5.964,149.333
C01367=1154.446,-68.667,-44.371,179.108,5.964,149.332
C01368=1154.441,-68.417,-44.382,179.110,5.965,149.332
C01369=1154.436,-68.167,-44.392,179.112,5.965,149.331
C01370=1154.430,-67.917,-44.402,179.114,5.965,149.331
C01371=1154.425,-67.668,-44.413,179.116,5.966,149.330
C01372=1154.420,-67.418,-44.424,179.119,5.966,149.329
C01373=1154.414,-67.169,-44.434,179.121,5.966,149.329
C01374=1154.409,-66.918,-44.445,179.123,5.967,149.328
C01375=1154.404,-66.669,-44.455,179.125,5.968,149.328
C01376=1154.399,-66.419,-44.466,179.128,5.968,149.327
C01377=1154.394,-66.170,-44.476,179.130,5.968,149.327
C01378=1154.388,-65.920,-44.487,179.132,5.969,149.326
C01379=1154.383,-65.670,-44.497,179.134,5.970,149.326
C01380=1154.378,-65.421,-44.508,179.137,5.970,149.325
C01381=1154.373,-65.171,-44.519,179.138,5.970,149.324
C01382=1154.367,-64.921,-44.529,179.141,5.970,149.324
C01383=1154.362,-64.671,-44.540,179.143,5.971,149.323
C01384=1154.357,-64.422,-44.550,179.145,5.972,149.323
C01385=1154.352,-64.172,-44.561,179.148,5.972,149.322
C01386=1154.346,-63.922,-44.571,179.150,5.972,149.322
C01387=1154.341,-63.673,-44.583,179.152,5.973,149.321
C01388=1154.336,-63.423,-44.593,179.155,5.973,149.320
C01389=1154.331,-63.173,-44.603,179.157,5.974,149.320
C01390=1154.325,-62.923,-44.614,179.159,5.974,149.319
C01391=1154.320,-62.673,-44.625,179.161,5.975,149.319
C01392=1154.314,-62.424,-44.636,179.164,5.975,149.318
C01393=1154.309,-62.174,-44.646,179.166,5.976,149.318
C01394=1154.304,-61.925,-44.657,179.169,5.976,149.317
C01395=1154.299,-61.674,-44.668,179.170,5.976,149.316
C01396=1154.294,-61.425,-44.679,179.172,5.977,149.316
C01397=1154.289,-61.175,-44.689,179.175,5.977,149.315
C01398=1154.283,-60.926,-44.699,179.177,5.978,149.315
C01399=1154.278,-60.676,-44.711,179.180,5.979,149.314
C01400=1154.272,-60.426,-44.721,179.181,5.979,149.313
C01401=1154.267,-60.177,-44.733,179.184,5.979,149.313
C01402=1154.262,-59.927,-44.743,179.186,5.980,149.312
C01403=1154.257,-59.677,-44.754,179.188,5.980,149.312
C01404=1154.252,-59.427,-44.765,179.191,5.981,149.311
C01405=1154.246,-59.178,-44.775,179.193,5.981,149.311
C01406=1154.241,-58.928,-44.787,179.195,5.981,149.310
C01407=1154.235,-58.678,-44.797,179.198,5.982,149.309
C01408=1154.231,-58.429,-44.808,179.200,5.983,149.309
C01409=1154.225,-58.179,-44.819,179.202,5.983,149.308
C01410=1154.220,-57.929,-44.830,179.204,5.983,149.308
C01411=1154.215,-57.679,-44.841,179.207,5.984,149.307
C01412=1154.209,-57.430,-44.852,179.209,5.984,149.307
C01413=1154.204,-57.180,-44.863,179.212,5.985,149.306
C01414=1154.199,-56.931,-44.874,179.214,5.986,149.305
C01415=1154.194,-56.680,-44.884,179.215,5.986,149.305
C01416=1154.189,-56.432,-44.895,179.218,5.986,149.304
C01417=1154.183,-56.181,-44.906,179.220,5.987,149.304
C01418=1154.178,-55.931,-44.917,179.223,5.987,149.303
C01419=1154.173,-55.682,-44.928,179.225,5.988,149.303
C01420=1154.168,-55.432,-44.939,179.227,5.988,149.302
C01421=1154.162,-55.182,-44.950,179.229,5.988,149.301
C01422=1154.157,-54.933,-44.961,179.232,5.989,149.301
C01423=1154.152,-54.682,-44.972,179.234,5.989,149.300
C01424=1154.147,-54.434,-44.983,179.236,5.990,149.300
C01425=1154.141,-54.184,-44.994,179.239,5.991,149.299
C01426=1154.136,-53.933,-45.005,179.241,5.991,149.299
C01427=1154.131,-53.684,-45.016,179.243,5.991,149.298
C01428=1154.126,-53.434,-45.027,179.245,5.992,149.297
C01429=1154.121,-53.184,-45.038,179.248,5.992,149.297
C01430=1154.115,-52.935,-45.049,179.250,5.993,149.296
C01431=1154.110,-52.685,-45.060,179.253,5.994,149.296
C01432=1154.104,-52.436,-45.071,179.255,5.993,149.295
C01433=1154.099,-52.186,-45.082,179.257,5.994,149.295
C01434=1154.095,-51.936,-45.093,179.259,5.995,149.294
C01435=1154.089,-51.687,-45.105,179.262,5.995,149.293
C01436=1154.084,-51.436,-45.115,179.264,5.996,149.293
C01437=1154.079,-51.187,-45.127,179.267,5.997,149.292
C01438=1154.073,-50.938,-45.138,179.269,5.996,149.291
C01439=1154.068,-50.667,-45.150,179.271,5.997,149.291
C01440=1154.062,-50.396,-45.162,179.273,5.997,149.290
C01441=1154.056,-50.126,-45.174,179.276,5.998,149.290
C01442=1154.051,-49.855,-45.186,179.278,5.999,149.289
C01443=1154.046,-49.605,-45.198,179.281,5.999,149.288
C01444=1154.040,-49.356,-45.209,179.283,6.000,149.288
C01445=1154.035,-49.106,-45.220,179.285,6.001,149.287
C01446=1154.030,-48.856,-45.231,179.288,6.001,149.287
C01447=1154.024,-48.607,-45.242,179.290,6.002,149.286
C01448=1154.019,-48.357,-45.254,179.292,6.001,149.286
C01449=1154.014,-48.107,-45.265,179.294,6.002,149.285
C01450=1154.008,-47.858,-45.276,179.297,6.003,149.284
C01451=1154.003,-47.608,-45.288,179.299,6.003,149.284
C01452=1153.998,-47.358,-45.299,179.302,6.004,149.283
C01453=1153.994,-47.108,-45.310,179.304,6.005,149.283
C01454=1153.987,-46.859,-45.321,179.307,6.005,149.282
C01455=1153.983,-46.609,-45.332,179.309,6.006,149.282
C01456=1153.977,-46.359,-45.344,179.311,6.006,149.281
C01457=1153.972,-46.109,-45.356,179.313,6.006,149.280
C01458=1153.966,-45.860,-45.367,179.315,6.007,149.280
C01459=1153.962,-45.611,-45.378,179.318,6.007,149.279
C01460=1153.956,-45.360,-45.390,179.320,6.008,149.279
C01461=1153.951,-45.110,-45.401,179.323,6.009,149.278
C01462=1153.946,-44.861,-45.412,179.325,6.009,149.278
C01463=1153.941,-44.612,-45.424,179.327,6.009,149.277
C01464=1153.936,-44.362,-45.435,179.329,6.010,149.276
C01465=1153.930,-44.112,-45.447,179.332,6.010,149.276
C01466=1153.925,-43.863,-45.458,179.334,6.011,149.275
C01467=1153.920,-43.613,-45.470,179.336,6.012,149.275
C01468=1153.915,-43.363,-45.480,179.339,6.012,149.274
C01469=1153.909,-43.113,-45.492,179.341,6.013,149.274
C01470=1153.904,-42.864,-45.503,179.344,6.013,149.273
C01471=1153.899,-42.614,-45.515,179.346,6.014,149.272
C01472=1153.894,-42.364,-45.526,179.348,6.014,149.272
C01473=1153.888,-42.114,-45.538,179.350,6.015,149.271
C01474=1153.883,-41.865,-45.550,179.353,6.015,149.270
C01475=1153.878,-41.616,-45.561,179.355,6.016,149.270
C01476=1153.872,-41.366,-45.573,179.358,6.016,149.269
C01477=1153.868,-41.116,-45.584,179.360,6.017,149.269
C01478=1153.862,-40.866,-45.596,179.362,6.018,149.268
C01479=1153.858,-40.617,-45.607,179.365,6.018,149.268
C01480=1153.852,-40.367,-45.619,179.367,6.019,149.267
C01481=1153.847,-40.118,-45.630,179.369,6.019,149.266
C01482=1153.841,-39.868,-45.642,179.371,6.019,149.266
C01483=1153.836,-39.618,-45.654,179.374,6.020,149.265
C01484=1153.831,-39.368,-45.665,179.376,6.021,149.265
C01485=1153.826,-39.118,-45.677,179.379,6.021,149.264
C01486=1153.821,-38.869,-45.688,179.381,6.022,149.264
C01487=1153.815,-38.619,-45.700,179.384,6.022,149.263
C01488=1153.810,-38.369,-45.712,179.386,6.023,149.262
C01489=1153.805,-38.120,-45.723,179.389,6.023,149.262
C01490=1153.800,-37.870,-45.735,179.391,6.024,149.261
C01491=1153.794,-37.620,-45.747,179.393,6.025,149.261
C01492=1153.790,-37.371,-45.759,179.395,6.025,149.260
C01493=1153.784,-37.122,-45.770,179.397,6.025,149.260
C01494=1153.778,-36.872,-45.782,179.400,6.026,149.259
C01495=1153.774,-36.622,-45.793,179.402,6.027,149.258
C01496=1153.768,-36.372,-45.805,179.405,6.027,149.258
C01497=1153.763,-36.122,-45.817,179.407,6.028,149.257
C01498=1153.758,-35.873,-45.828,179.410,6.028,149.257
C01499=1153.753,-35.623,-45.840,179.412,6.029,149.256
C01500=1153.747,-35.373,-45.853,179.414,6.029,149.255
C01501=1153.743,-35.124,-45.864,179.417,6.030,149.255
C01502=1153.737,-34.875,-45.876,179.419,6.031,149.254
C01503=1153.731,-34.625,-45.888,179.421,6.031,149.254
C01504=1153.727,-34.375,-45.899,179.424,6.032,149.253
C01505=1153.721,-34.125,-45.911,179.426,6.032,149.253
C01506=1153.716,-33.876,-45.923,179.428,6.032,149.252
C01507=1153.711,-33.626,-45.935,179.431,6.033,149.251
C01508=1153.706,-33.376,-45.947,179.433,6.033,149.251
C01509=1153.701,-33.126,-45.959,179.435,6.034,149.250
C01510=1153.695,-32.877,-45.971,179.438,6.035,149.250
C01511=1153.691,-32.627,-45.982,179.440,6.035,149.249
C01512=1153.685,-32.377,-45.994,179.442,6.036,149.249
C01513=1153.680,-32.127,-46.006,179.445,6.037,149.248
C01514=1153.675,-31.878,-46.019,179.447,6.037,149.247
C01515=1153.669,-31.628,-46.031,179.450,6.038,149.247
C01516=1153.664,-31.379,-46.042,179.452,6.039,149.246
C01517=1153.659,-31.129,-46.053,179.455,6.039,149.246
C01518=1153.653,-30.880,-46.066,179.457,6.040,149.245
C01519=1153.648,-30.630,-46.078,179.460,6.040,149.244
C01520=1153.643,-30.380,-46.089,179.462,6.041,149.244
C01521=1153.638,-30.131,-46.102,179.464,6.042,149.243
C01522=1153.633,-29.881,-46.114,179.467,6.042,149.243
C01523=1153.627,-29.631,-46.126,179.469,6.042,149.242
C01524=1153.622,-29.382,-46.138,179.471,6.043,149.242
C01525=1153.618,-29.132,-46.150,179.474,6.043,149.241
C01526=1153.612,-28.882,-46.161,179.476,6.044,149.240
C01527=1153.607,-28.633,-46.174,179.478,6.044,149.240
C01528=1153.602,-28.383,-46.186,179.481,6.045,149.239
C01529=1153.596,-28.134,-46.198,179.483,6.046,149.239
C01530=1153.591,-27.884,-46.210,179.485,6.046,149.238
C01531=1153.586,-27.634,-46.222,179.488,6.047,149.238
C01532=1153.581,-27.385,-46.234,179.490,6.048,149.237
C01533=1153.576,-27.135,-46.246,179.492,6.048,149.236
C01534=1153.571,-26.886,-46.259,179.495,6.049,149.236
C01535=1153.565,-26.636,-46.271,179.497,6.050,149.235
C01536=1153.560,-26.386,-46.283,179.500,6.050,149.235
C01537=1153.555,-26.136,-46.295,179.502,6.051,149.234
C01538=1153.550,-25.886,-46.307,179.505,6.051,149.233
C01539=1153.545,-25.637,-46.319,179.507,6.052,149.233
C01540=1153.540,-25.387,-46.331,179.510,6.053,149.232
C01541=1153.535,-25.138,-46.344,179.512,6.053,149.232
C01542=1153.529,-24.888,-46.356,179.514,6.054,149.231
C01543=1153.524,-24.619,-46.369,179.517,6.055,149.231
C01544=1153.518,-24.348,-46.383,179.519,6.055,149.230
C01545=1153.512,-24.078,-46.396,179.522,6.055,149.229
C01546=1153.507,-23.809,-46.409,179.525,6.057,149.229
C01547=1153.501,-23.559,-46.421,179.527,6.057,149.228
C01548=1153.496,-23.309,-46.433,179.530,6.058,149.228
C01549=1153.491,-23.059,-46.446,179.532,6.059,149.227
C01550=1153.486,-22.809,-46.458,179.534,6.059,149.226
C01551=1153.481,-22.559,-46.470,179.537,6.060,149.226
C01552=1153.476,-22.310,-46.483,179.539,6.061,149.225
C01553=1153.471,-22.061,-46.495,179.542,6.061,149.225
C01554=1153.465,-21.811,-46.507,179.544,6.062,149.224
C01555=1153.460,-21.561,-46.520,179.547,6.062,149.223
C01556=1153.455,-21.312,-46.532,179.549,6.063,149.223
C01557=1153.450,-21.062,-46.544,179.552,6.064,149.222
C01558=1153.444,-20.813,-46.557,179.554,6.064,149.222
C01559=1153.440,-20.562,-46.569,179.557,6.065,149.221
C01560=1153.434,-20.313,-46.582,179.559,6.066,149.221
C01561=1153.429,-20.063,-46.594,179.561,6.066,149.220
C01562=1153.424,-19.814,-46.606,179.564,6.067,149.219
C01563=1153.419,-19.564,-46.619,179.566,6.067,149.219
C01564=1153.413,-19.314,-46.631,179.568,6.068,149.218
C01565=1153.408,-19.065,-46.643,179.571,6.068,149.218
C01566=1153.403,-18.816,-46.656,179.573,6.069,149.217
C01567=1153.398,-18.565,-46.668,179.576,6.070,149.216
C01568=1153.392,-18.316,-46.681,179.578,6.071,149.216
C01569=1153.387,-18.066,-46.694,179.581,6.071,149.215
C01570=1153.382,-17.817,-46.707,179.583,6.072,149.215
C01571=1153.377,-17.567,-46.718,179.586,6.072,149.214
C01572=1153.372,-17.318,-46.731,179.588,6.073,149.214
C01573=1153.367,-17.068,-46.744,179.590,6.073,149.213
C01574=1153.362,-16.818,-46.757,179.593,6.074,149.212
C01575=1153.357,-16.568,-46.769,179.595,6.075,149.212
C01576=1153.351,-16.319,-46.781,179.597,6.075,149.211
C01577=1153.346,-16.070,-46.794,179.600,6.076,149.211
C01578=1153.341,-15.819,-46.807,179.602,6.077,149.210
C01579=1153.336,-15.569,-46.819,179.605,6.077,149.209
C01580=1153.331,-15.320,-46.832,179.607,6.078,149.209
C01581=1153.325,-15.071,-46.844,179.609,6.079,149.208
C01582=1153.320,-14.822,-46.857,179.612,6.079,149.208
C01583=1153.316,-14.571,-46.870,179.614,6.080,149.207
C01584=1153.310,-14.322,-46.882,179.617,6.080,149.207
C01585=1153.304,-14.072,-46.895,179.619,6.081,149.206
C01586=1153.299,-13.823,-46.908,179.622,6.082,149.205
C01587=1153.294,-13.573,-46.920,179.624,6.082,149.205
C01588=1153.290,-13.323,-46.933,179.626,6.083,149.204
C01589=1153.285,-13.074,-46.946,179.629,6.084,149.204
C01590=1153.279,-12.825,-46.958,179.632,6.085,149.203
C01591=1153.274,-12.575,-46.972,179.634,6.086,149.203
C01592=1153.269,-12.324,-46.984,179.637,6.086,149.202
C01593=1153.264,-12.075,-46.996,179.639,6.087,149.201
C01594=1153.258,-11.826,-47.009,179.642,6.087,149.201
C01595=1153.253,-11.576,-47.022,179.644,6.088,149.200
C01596=1153.248,-11.326,-47.035,179.646,6.089,149.200
C01597=1153.243,-11.077,-47.048,179.649,6.089,149.199
C01598=1153.238,-10.827,-47.060,179.651,6.090,149.198
C01599=1153.233,-10.577,-47.073,179.653,6.091,149.198
C01600=1153.227,-10.328,-47.087,179.656,6.091,149.197
C01601=1153.222,-10.078,-47.099,179.658,6.092,149.197
C01602=1153.217,-9.829,-47.112,179.661,6.092,149.196
C01603=1153.212,-9.579,-47.125,179.663,6.093,149.196
C01604=1153.207,-9.330,-47.138,179.666,6.094,149.195
C01605=1153.202,-9.080,-47.151,179.668,6.095,149.195
C01606=1153.197,-8.830,-47.163,179.671,6.096,149.194
C01607=1153.191,-8.581,-47.177,179.673,6.096,149.193
C01608=1153.186,-8.331,-47.189,179.676,6.097,149.193
C01609=1153.182,-8.081,-47.202,179.678,6.098,149.192
C01610=1153.176,-7.832,-47.215,179.681,6.098,149.192
C01611=1153.171,-7.582,-47.228,179.683,6.099,149.191
C01612=1153.166,-7.332,-47.241,179.686,6.099,149.190
C01613=1153.160,-7.083,-47.254,179.688,6.100,149.190
C01614=1153.155,-6.833,-47.267,179.690,6.101,149.189
C01615=1153.151,-6.583,-47.280,179.693,6.101,149.189
C01616=1153.145,-6.334,-47.293,179.696,6.103,149.188
C01617=1153.140,-6.085,-47.306,179.698,6.103,149.188
C01618=1153.135,-5.835,-47.319,179.701,6.104,149.187
C01619=1153.130,-5.585,-47.332,179.703,6.105,149.186
C01620=1153.124,-5.336,-47.345,179.706,6.105,149.186
C01621=1153.120,-5.086,-47.358,179.708,6.106,149.185
C01622=1153.114,-4.836,-47.371,179.710,6.106,149.185
C01623=1153.109,-4.587,-47.384,179.713,6.107,149.184
C01624=1153.104,-4.337,-47.398,179.715,6.108,149.183
C01625=1153.099,-4.088,-47.411,179.717,6.108,149.183
C01626=1153.094,-3.838,-47.424,179.720,6.110,149.183
C01627=1153.089,-3.588,-47.437,179.723,6.111,149.182
C01628=1153.083,-3.339,-47.449,179.725,6.111,149.181
C01629=1153.078,-3.089,-47.463,179.728,6.112,149.181
C01630=1153.073,-2.840,-47.476,179.730,6.113,149.180
C01631=1153.068,-2.590,-47.490,179.732,6.113,149.180
C01632=1153.063,-2.340,-47.502,179.735,6.114,149.179
C01633=1153.058,-2.091,-47.515,179.737,6.114,149.178
C01634=1153.053,-1.841,-47.529,179.739,6.115,149.178
C01635=1153.048,-1.592,-47.542,179.743,6.116,149.177
C01636=1153.042,-1.342,-47.556,179.745,6.117,149.177
C01637=1153.037,-1.092,-47.568,179.748,6.118,149.176
C01638=1153.032,-0.843,-47.582,179.750,6.118,149.176
C01639=1153.027,-0.593,-47.595,179.752,6.119,149.175
C01640=1153.021,-0.344,-47.608,179.755,6.120,149.174
C01641=1153.017,-0.094,-47.622,179.757,6.120,149.174
C01642=1153.011,0.155,-47.635,179.759,6.121,149.173
C01643=1153.007,0.405,-47.648,179.763,6.122,149.173
C01644=1153.001,0.654,-47.662,179.765,6.123,149.172
C01645=1152.997,0.904,-47.675,179.767,6.123,149.171
C01646=1152.991,1.154,-47.688,179.770,6.124,149.171
C01647=1152.985,1.423,-47.703,179.772,6.125,149.170
C01648=1152.980,1.693,-47.717,179.776,6.126,149.170
C01649=1152.974,1.962,-47.731,179.778,6.127,149.169
C01650=1152.969,2.231,-47.746,179.780,6.127,149.168
C01651=1152.964,2.481,-47.759,179.783,6.128,149.168
C01652=1152.959,2.731,-47.773,179.786,6.129,149.167
C01653=1152.954,2.980,-47.786,179.788,6.130,149.167
C01654=1152.948,3.230,-47.799,179.791,6.131,149.166
C01655=1152.943,3.479,-47.813,179.793,6.131,149.166
C01656=1152.938,3.729,-47.826,179.795,6.132,149.165
C01657=1152.933,3.978,-47.840,179.798,6.133,149.165
C01658=1152.928,4.228,-47.853,179.800,6.133,149.164
C01659=1152.923,4.478,-47.867,179.803,6.135,149.163
C01660=1152.918,4.727,-47.881,179.806,6.135,149.163
C01661=1152.913,4.977,-47.894,179.808,6.136,149.162
C01662=1152.907,5.226,-47.908,179.811,6.136,149.162
C01663=1152.902,5.477,-47.921,179.813,6.137,149.161
C01664=1152.897,5.725,-47.934,179.815,6.138,149.160
C01665=1152.892,5.976,-47.948,179.818,6.139,149.160
C01666=1152.887,6.224,-47.961,179.821,6.140,149.159
C01667=1152.882,6.475,-47.975,179.823,6.141,149.159
C01668=1152.876,6.724,-47.989,179.826,6.141,149.158
C01669=1152.872,6.973,-48.002,179.828,6.142,149.158
C01670=1152.867,7.223,-48.016,179.830,6.142,149.157
C01671=1152.861,7.472,-48.030,179.833,6.144,149.156
C01672=1152.857,7.723,-48.043,179.836,6.144,149.156
C01673=1152.851,7.972,-48.057,179.838,6.145,149.155
C01674=1152.846,8.222,-48.070,179.841,6.146,149.155
C01675=1152.841,8.471,-48.084,179.843,6.146,149.154
C01676=1152.836,8.720,-48.098,179.846,6.148,149.154
C01677=1152.831,8.971,-48.112,179.848,6.148,149.153
C01678=1152.826,9.220,-48.125,179.851,6.149,149.152
C01679=1152.821,9.469,-48.139,179.853,6.150,149.152
C01680=1152.815,9.719,-48.152,179.856,6.150,149.151
C01681=1152.810,9.968,-48.167,179.859,6.152,149.151
C01682=1152.806,10.218,-48.181,179.861,6.152,149.150
C01683=1152.800,10.467,-48.193,179.863,6.153,149.150
C01684=1152.795,10.717,-48.208,179.866,6.154,149.149
C01685=1152.790,10.966,-48.222,179.868,6.154,149.148
C01686=1152.785,11.216,-48.235,179.871,6.156,149.148
C01687=1152.780,11.466,-48.250,179.874,6.156,149.147
C01688=1152.775,11.715,-48.263,179.876,6.157,149.147
C01689=1152.770,11.965,-48.276,179.878,6.158,149.146
C01690=1152.765,12.215,-48.291,179.881,6.159,149.146
C01691=1152.759,12.464,-48.305,179.884,6.160,149.145
C01692=1152.754,12.714,-48.319,179.886,6.161,149.145
C01693=1152.750,12.964,-48.332,179.889,6.161,149.144
C01694=1152.744,13.213,-48.346,179.891,6.162,149.143
C01695=1152.739,13.462,-48.360,179.893,6.162,149.143
C01696=1152.734,13.712,-48.374,179.896,6.164,149.142
C01697=1152.728,13.962,-48.387,179.899,6.164,149.142
C01698=1152.723,14.211,-48.402,179.901,6.165,149.141
C01699=1152.719,14.461,-48.415,179.904,6.166,149.140
C01700=1152.714,14.710,-48.429,179.906,6.167,149.140
C01701=1152.709,14.959,-48.444,179.909,6.168,149.139
C01702=1152.704,15.209,-48.458,179.911,6.169,149.139
C01703=1152.698,15.459,-48.471,179.914,6.169,149.138
C01704=1152.693,15.709,-48.485,179.916,6.170,149.138
C01705=1152.688,15.958,-48.500,179.919,6.171,149.137
C01706=1152.682,16.207,-48.514,179.922,6.172,149.137
C01707=1152.678,16.457,-48.527,179.924,6.173,149.136
C01708=1152.673,16.706,-48.542,179.926,6.173,149.135
C01709=1152.668,16.956,-48.556,179.929,6.175,149.135
C01710=1152.663,17.205,-48.570,179.932,6.175,149.134
C01711=1152.658,17.455,-48.584,179.934,6.176,149.134
C01712=1152.652,17.705,-48.598,179.937,6.177,149.133
C01713=1152.647,17.955,-48.612,179.939,6.178,149.133
C01714=1152.642,18.204,-48.626,179.942,6.179,149.132
C01715=1152.637,18.454,-48.640,179.944,6.180,149.132
C01716=1152.632,18.703,-48.654,179.947,6.180,149.131
C01717=1152.627,18.953,-48.669,179.950,6.182,149.130
C01718=1152.621,19.202,-48.682,179.952,6.182,149.130
C01719=1152.617,19.452,-48.697,179.954,6.183,149.129
C01720=1152.612,19.701,-48.711,179.957,6.183,149.129
C01721=1152.607,19.951,-48.725,179.960,6.185,149.128
C01722=1152.601,20.200,-48.739,179.962,6.185,149.127
C01723=1152.596,20.450,-48.754,179.965,6.186,149.127
C01724=1152.591,20.700,-48.768,179.967,6.187,149.126
C01725=1152.586,20.949,-48.782,179.970,6.188,149.126
C01726=1152.581,21.199,-48.796,179.972,6.189,149.125
C01727=1152.576,21.448,-48.810,179.975,6.190,149.125
C01728=1152.571,21.698,-48.825,179.977,6.190,149.124
C01729=1152.566,21.947,-48.840,179.980,6.192,149.124
C01730=1152.561,22.196,-48.854,179.982,6.193,149.123
C01731=1152.556,22.446,-48.868,179.985,6.193,149.122
C01732=1152.551,22.695,-48.882,179.987,6.194,149.122
C01733=1152.546,22.945,-48.896,179.991,6.195,149.121
C01734=1152.541,23.195,-48.911,179.993,6.196,149.121
C01735=1152.536,23.444,-48.925,179.995,6.196,149.120
C01736=1152.531,23.694,-48.939,179.998,6.198,149.120
C01737=1152.526,23.944,-48.953,-179.999,6.198,149.119
C01738=1152.520,24.192,-48.969,-179.997,6.199,149.119
C01739=1152.515,24.442,-48.983,-179.994,6.200,149.118
C01740=1152.510,24.692,-48.997,-179.992,6.201,149.117
C01741=1152.505,24.942,-49.011,-179.990,6.202,149.117
C01742=1152.500,25.191,-49.026,-179.987,6.203,149.116
C01743=1152.495,25.440,-49.041,-179.984,6.204,149.116
C01744=1152.490,25.690,-49.055,-179.981,6.205,149.115
C01745=1152.485,25.939,-49.069,-179.979,6.206,149.115
C01746=1152.479,26.189,-49.084,-179.977,6.206,149.114
C01747=1152.474,26.439,-49.098,-179.974,6.208,149.114
C01748=1152.470,26.688,-49.113,-179.971,6.208,149.113
C01749=1152.465,26.938,-49.127,-179.969,6.209,149.112
C01750=1152.460,27.187,-49.142,-179.966,6.210,149.112
C01751=1152.455,27.456,-49.157,-179.964,6.211,149.111
C01752=1152.449,27.725,-49.174,-179.960,6.212,149.111
C01753=1152.444,27.994,-49.189,-179.958,6.213,149.110
C01754=1152.438,28.263,-49.204,-179.955,6.214,149.110
C01755=1152.432,28.512,-49.220,-179.952,6.215,149.109
C01756=1152.427,28.762,-49.234,-179.950,6.216,149.108
C01757=1152.422,29.012,-49.248,-179.947,6.217,149.108
C01758=1152.418,29.261,-49.263,-179.945,6.218,149.107
C01759=1152.413,29.510,-49.277,-179.942,6.218,149.107
C01760=1152.407,29.760,-49.292,-179.939,6.220,149.106
C01761=1152.402,30.010,-49.307,-179.937,6.221,149.106
C01762=1152.397,30.259,-49.321,-179.935,6.221,149.105
C01763=1152.393,30.508,-49.336,-179.932,6.222,149.105
C01764=1152.387,30.758,-49.351,-179.929,6.223,149.104
C01765=1152.382,31.008,-49.366,-179.927,6.224,149.103
C01766=1152.377,31.257,-49.381,-179.924,6.225,149.103
C01767=1152.372,31.507,-49.395,-179.922,6.226,149.102
C01768=1152.367,31.756,-49.410,-179.919,6.227,149.102
C01769=1152.362,32.006,-49.425,-179.917,6.228,149.101
C01770=1152.357,32.255,-49.440,-179.914,6.229,149.101
C01771=1152.352,32.505,-49.455,-179.911,6.230,149.100
C01772=1152.347,32.755,-49.469,-179.909,6.231,149.100
C01773=1152.342,33.004,-49.484,-179.906,6.232,149.099
C01774=1152.336,33.254,-49.499,-179.904,6.233,149.098
C01775=1152.332,33.503,-49.514,-179.901,6.233,149.098
C01776=1152.327,33.753,-49.528,-179.898,6.235,149.097
C01777=1152.321,34.002,-49.544,-179.896,6.235,149.097
C01778=1152.317,34.252,-49.558,-179.893,6.237,149.096
C01779=1152.312,34.501,-49.573,-179.890,6.237,149.096
C01780=1152.306,34.750,-49.588,-179.888,6.238,149.095
C01781=1152.302,35.000,-49.603,-179.885,6.240,149.095
C01782=1152.296,35.249,-49.618,-179.883,6.240,149.094
C01783=1152.291,35.499,-49.633,-179.881,6.241,149.094
C01784=1152.287,35.748,-49.648,-179.877,6.242,149.093
C01785=1152.281,35.998,-49.662,-179.875,6.243,149.092
C01786=1152.276,36.247,-49.677,-179.873,6.244,149.092
C01787=1152.271,36.497,-49.693,-179.870,6.245,149.091
C01788=1152.266,36.746,-49.707,-179.867,6.246,149.091
C01789=1152.261,36.996,-49.722,-179.865,6.247,149.090
C01790=1152.255,37.246,-49.737,-179.862,6.248,149.090
C01791=1152.251,37.495,-49.752,-179.860,6.249,149.089
C01792=1152.245,37.744,-49.768,-179.857,6.250,149.089
C01793=1152.241,37.994,-49.782,-179.854,6.251,149.088
C01794=1152.235,38.243,-49.798,-179.852,6.252,149.087
C01795=1152.230,38.492,-49.813,-179.849,6.253,149.087
C01796=1152.225,38.743,-49.828,-179.847,6.254,149.086
C01797=1152.221,38.992,-49.843,-179.844,6.254,149.086
C01798=1152.215,39.241,-49.858,-179.841,6.256,149.085
C01799=1152.211,39.491,-49.873,-179.839,6.257,149.085
C01800=1152.205,39.741,-49.888,-179.836,6.258,149.084
C01801=1152.200,39.990,-49.903,-179.834,6.259,149.084
C01802=1152.195,40.239,-49.919,-179.831,6.259,149.083
C01803=1152.190,40.489,-49.933,-179.828,6.261,149.083
C01804=1152.185,40.738,-49.949,-179.826,6.262,149.082
C01805=1152.181,40.988,-49.964,-179.823,6.263,149.081
C01806=1152.175,41.237,-49.980,-179.821,6.264,149.081
C01807=1152.171,41.486,-49.995,-179.818,6.264,149.080
C01808=1152.165,41.736,-50.010,-179.815,6.266,149.080
C01809=1152.160,41.986,-50.025,-179.813,6.267,149.079
C01810=1152.155,42.235,-50.040,-179.810,6.268,149.079
C01811=1152.150,42.484,-50.055,-179.807,6.269,149.078
C01812=1152.145,42.734,-50.071,-179.805,6.270,149.078
C01813=1152.140,42.984,-50.087,-179.802,6.271,149.077
C01814=1152.135,43.233,-50.101,-179.800,6.272,149.076
C01815=1152.130,43.483,-50.117,-179.797,6.273,149.076
C01816=1152.125,43.732,-50.132,-179.794,6.274,149.075
C01817=1152.120,43.981,-50.147,-179.792,6.275,149.075
C01818=1152.115,44.231,-50.163,-179.789,6.276,149.074
C01819=1152.110,44.480,-50.178,-179.787,6.277,149.074
C01820=1152.105,44.730,-50.194,-179.784,6.278,149.073
C01821=1152.100,44.979,-50.209,-179.781,6.279,149.073
C01822=1152.095,45.228,-50.224,-179.779,6.281,149.072
C01823=1152.090,45.478,-50.240,-179.776,6.281,149.072
C01824=1152.085,45.728,-50.254,-179.774,6.282,149.071
C01825=1152.080,45.977,-50.270,-179.771,6.283,149.070
C01826=1152.074,46.227,-50.286,-179.768,6.284,149.070
C01827=1152.070,46.477,-50.301,-179.766,6.286,149.070
C01828=1152.065,46.726,-50.317,-179.763,6.286,149.069
C01829=1152.059,46.975,-50.332,-179.760,6.288,149.068
C01830=1152.055,47.225,-50.347,-179.758,6.288,149.068
C01831=1152.049,47.474,-50.363,-179.756,6.289,149.067
C01832=1152.045,47.724,-50.379,-179.752,6.290,149.067
C01833=1152.039,47.973,-50.394,-179.750,6.291,149.066
C01834=1152.035,48.222,-50.410,-179.747,6.293,149.066
C01835=1152.030,48.472,-50.426,-179.745,6.293,149.065
C01836=1152.025,48.721,-50.442,-179.742,6.295,149.065
C01837=1152.020,48.971,-50.457,-179.739,6.295,149.064
C01838=1152.015,49.220,-50.472,-179.737,6.297,149.064
C01839=1152.010,49.470,-50.488,-179.734,6.298,149.063
C01840=1152.004,49.719,-50.504,-179.732,6.298,149.062
C01841=1152.000,49.969,-50.519,-179.729,6.300,149.062
